# B&R Automation Studio project NAELD004C00R10L518F00 (part 42)

#### Act_Background_QueryWorkOrderInfo.st
```iecst
(** 2021-08-01 **)
ACTION Act_Background_QueryWorkOrderInfo:

	IF eStatus2 <> Error THEN
		IF  uiMilliSecOld <> p_tyDTStructure.millisec THEN
			IF EDGEPOS(p_bLinkOpsMagConvLD1QueryWO) THEN //query false when rcp loaded
				sMagazineId 		:= '1'; //Magazine position to mes
				bGUIDInserted[1]	:= FALSE;
				a_bQueryQueue[i2] 	:= TRUE;
				i2 := i2 + 1;
			ELSIF EDGEPOS(p_bLinkOpsMagConvLD2QueryWO) THEN
				sMagazineId 		:= '2';
				bGUIDInserted[2]	:= FALSE;
				a_bQueryQueue[i2] 	:= TRUE;
				i2 := i2 + 1;
			ELSIF EDGEPOS(p_bLinkOpsMagConvLD3QueryWO) THEN
				sMagazineId 		:= '3';
				bGUIDInserted[3]	:= FALSE;
				a_bQueryQueue[i2] 	:= TRUE;
				i2 := i2 + 1;
			END_IF
		END_IF

//		IF EDGEPOS(p_bQueryWorkOrderInfo) AND p_bAcceptCondition THEN
//		IF (EDGEPOS((p_eLinkCustomerReq = Siemens AND p_bOpsConvWaitForTopUpBrd OR (p_usiLinkProdRcpCurrRcpMcMod = 0 AND bQueryloaderWorkOrder = FALSE) AND bConnected AND p_bOpsRun) AND p_bQueryWorkOrderInfo = FALSE AND bManualQueryWO = FALSE AND p_eLinkCustomerReq = NA)  (*AND p_bAcceptCondition*) AND bReplyWorkOrderInfo= FALSE AND sWorkOrderId = ''))
//			 OR EDGEPOS (p_bQueryWorkOrderInfo) THEN        //Query For Loader           //ADD
//		IF (EDGEPOS((p_bSiemensMcModeChgPrep AND (p_bOpsConvWaitForTopUpBrd OR p_usiLinkProdRcpCurrRcpMcMod = 0)  AND bQueryloaderWorkOrder = FALSE AND bConnected AND p_bOpsRun) AND p_bQueryWorkOrderInfo = FALSE AND bManualQueryWO = FALSE AND bReplyWorkOrderInfo= FALSE AND sWorkOrderId = ''))
//			 OR EDGEPOS (p_bQueryWorkOrderInfo) THEN        //Query For Loader           //ADD
//		IF bQueryloaderWorkOrder = FALSE AND bConnected AND p_bOpsRun AND p_bQueryWorkOrderInfo = FALSE AND bManualQueryWO = FALSE AND bReplyWorkOrderInfo= FALSE AND sWorkOrderId = ''
//			OR EDGEPOS (p_bQueryWorkOrderInfo) THEN        //Query For Loader           //ADD
		IF bQueryloaderWorkOrder = FALSE AND bConnected AND p_bOpsRun AND p_bQueryWorkOrderInfo = FALSE AND bManualQueryWO = FALSE AND bReplyWorkOrderInfo= FALSE AND sWorkOrderId = ''
			OR a_bQueryQueue[0]  THEN
			//OR EDGEPOS (p_bLinkOpsMagConvLD1QueryWO) OR EDGEPOS (p_bLinkOpsMagConvLD2QueryWO) OR EDGEPOS (p_bLinkOpsMagConvLD3QueryWO) THEN        //Query For Loader           //ADD

			fHermesAddOneMsgSend(ADR(a_eMsgSend) , ADR(udiMsgSendBffr) , HermesMsgTypeQueryWorkOrderInfo);

			fHermesGenerateUUID(ADR(tyQueryWorkOrderInfo.tyData.sQueryId) , p_tyDTStructure , pa_usiMacAddr); //Generate QueryID
			uiMilliSecOld :=  p_tyDTStructure.millisec;

			tyQueryWorkOrderInfo.tyData.sMachineId							:= p_sMcId;
			IF sMagazineId = '1'  AND bGUIDInserted[1] = FALSE THEN //Magazine position to mes
				a_MagGUID[1] 		:= tyQueryWorkOrderInfo.tyData.sQueryId;
				bGUIDInserted[1] 	:= TRUE;
			ELSIF sMagazineId = '2' AND bGUIDInserted[2] = FALSE THEN
				a_MagGUID[2] 		:= tyQueryWorkOrderInfo.tyData.sQueryId;
				bGUIDInserted[2] 	:= TRUE;
			ELSIF sMagazineId = '3' AND bGUIDInserted[3] = FALSE THEN
				a_MagGUID[3] 		:= tyQueryWorkOrderInfo.tyData.sQueryId;
				bGUIDInserted[3] 	:= TRUE;
			END_IF

			memcpy(ADR(a_bQueryQueue[0]) , ADR(a_bQueryQueue[1]) , SIZEOF(a_bQueryQueue[0]) * 3);
			a_bQueryQueue[3]	:= FALSE;
			i2 := i2 - 1;

			tyQueryWorkOrderInfo.tyData.sMagazineId							:= p_sMagazineId;
			tyQueryWorkOrderInfo.tyData.iSlotId								:= p_iSlotId;
			tyQueryWorkOrderInfo.tyData.sBarcode						    := p_sBarcode;
			tyQueryWorkOrderInfo.tyAvl.bQueryId							    := tyQueryWorkOrderInfo.tyData.sQueryId <> '';
			tyQueryWorkOrderInfo.tyAvl.bMachineId							:= tyQueryWorkOrderInfo.tyData.sMachineId <> '';
			tyQueryWorkOrderInfo.tyAvl.bMagazineId							:= tyQueryWorkOrderInfo.tyData.sMagazineId <> '';
			tyQueryWorkOrderInfo.tyAvl.bSlotId								:= tyQueryWorkOrderInfo.tyData.iSlotId <> 0;
			tyQueryWorkOrderInfo.tyAvl.bBarcode								:= tyQueryWorkOrderInfo.tyData.sBarcode <> '';

			bQueryloaderWorkOrder := TRUE;
			bRcvWorkOrderInfo1 := FALSE;                     //ADD
			bRcvWorkOrderInfo2 := FALSE;
			bSndWorkOrderInfo  := FALSE;

		END_IF
		                                                                      //Reply Bypass Workorder
//		IF EDGEPOS((p_bSiemensMcModeChgPrep AND bConnected AND p_bOpsRun) AND bReplyBypassWorkOrderInfo= FALSE AND p_bUSHermesUSRdy AND bNewIncomingBoard)  THEN        //Query For Bypass mode           //ADD
//
//
//			fHermesAddOneMsgSend(ADR(a_eMsgSend) , ADR(udiMsgSendBffr) , HermesMsgTypeQueryBypassWOInfo);
//
//			fHermesGenerateUUID(ADR(tyQueryBypassWorkOrderInfo.tyData.sQueryId) , p_tyDTStructure , pa_usiMacAddr); //Generate QueryID
//
//			tyQueryBypassWorkOrderInfo.tyData.sMachineId							:= p_sMcId;
//			tyQueryBypassWorkOrderInfo.tyData.sMagazineId							:= p_sMagazineId;
//			tyQueryBypassWorkOrderInfo.tyData.iSlotId								:= p_iSlotId;
//			tyQueryBypassWorkOrderInfo.tyData.sBarcode						        := sUSBarcode;
//
//			tyQueryBypassWorkOrderInfo.tyAvl.bQueryId							    := tyQueryBypassWorkOrderInfo.tyData.sQueryId <> '';
//			tyQueryBypassWorkOrderInfo.tyAvl.bMachineId						     	:= tyQueryBypassWorkOrderInfo.tyData.sMachineId <> '';
//			tyQueryBypassWorkOrderInfo.tyAvl.bMagazineId							:= tyQueryBypassWorkOrderInfo.tyData.sMagazineId <> '';
//			tyQueryBypassWorkOrderInfo.tyAvl.bSlotId								:= tyQueryBypassWorkOrderInfo.tyData.iSlotId <> 0;
//			tyQueryBypassWorkOrderInfo.tyAvl.bBarcode								:= tyQueryBypassWorkOrderInfo.tyData.sBarcode <> '';
//
//			bQueryBypassWorkOrder := TRUE;
//			bRcvWorkBypassOrderInfo := FALSE;
//			bRcvBypassWorkOrderInfo2 := FALSE;
//			bRcvWorkOrderInfo3      :=FALSE;
//		END_IF

		IF p_bQueryWorkOrderInfo AND p_bAcceptCondition =FALSE THEN
			bRstWorkOrderInfo := TRUE;
		END_IF

		IF tyMsgTypeRcv.bSendWorkOrderInfo THEN

//			IF p_bQueryWorkOrderInfo AND (udiStatus2 = 0) THEN //After CmpParamRcv
//			IF (p_bQueryWorkOrderInfo OR p_bOpsConvWaitForTopUpBrd) AND (udiStatus2 = 0) AND p_tyDI.bTopCoverSWSig THEN //After CmpParamRcv
			IF (p_bQueryWorkOrderInfo OR p_eLinkCustomerReq = Siemens) AND (udiStatus2 = 0) THEN //After CmpParamRcv
				IF tySendWorkOrderInfoRcv.tyAvl.bWorkOrderId AND tySendWorkOrderInfoRcv.tyData.sWorkOrderId <> '' AND
				   tySendWorkOrderInfoRcv.tyData.rWidth >= 50.0 AND tySendWorkOrderInfoRcv.tyData.rWidth <= 460.0	(*AND p_bAcceptCondition*) THEN //Wait Accept Conditon On

					//Priority setting
					memset(ADR(usiSum),0,SIZEOF(usiSum));
					FOR i := 1 TO 3 DO
						usiSum[i]	:= usiSum[i] + usiMagPrior[i];
						IF a_MagGUID[i] = tySendWorkOrderInfoRcv.tyData.sQueryId THEN
							usiSum[i] := usiSum[i] + 10;
						END_IF
					END_FOR
					FOR i1:=1 TO 3 DO
						//Assign Magazine order
						IF  usiSum[i1] >=10 THEN
							IF a_MagAccOrder[1]=0 AND a_MagAccOrder[2]=0 AND a_MagAccOrder[3]=0 THEN
								a_MagAccOrder[i1] := 10; //output
								usiMagOrderPos := i1;
							ELSIF ((a_MagAccOrder[1]=0 AND a_MagAccOrder[2]=0) OR
								(a_MagAccOrder[2]=0 AND a_MagAccOrder[3]=0) OR
								(a_MagAccOrder[1]=0 AND a_MagAccOrder[3]=0)) AND a_MagAccOrder[i1] =0 THEN
								a_MagAccOrder[i1] := 20;
								usiMagOrderPos := i1;
							ELSIF (a_MagAccOrder[1]=0 OR a_MagAccOrder[2]=0 OR a_MagAccOrder[3]=0) AND a_MagAccOrder[i1] =0 THEN
								a_MagAccOrder[i1] := 30;
								usiMagOrderPos := i1;
							END_IF
							bGUIDInserted[i1] := FALSE;
						END_IF
					END_FOR

					bSndWorkOrderInfo  := TRUE;
					bRcvWorkOrderInfo1 := TRUE;
					bRetainNewAcc      := FALSE;                            //ADD
					bQueryloaderWorkOrder := FALSE;
					tySendWorkOrderInfoAcc := tySendWorkOrderInfoRcv;
					tyMsgTypeRcv.bSendWorkOrderInfo := FALSE;
					sWorkOrderId := tySendWorkOrderInfoRcv.tyData.sWorkOrderId;

				ELSIF (tySendWorkOrderInfoRcv.tyAvl.bWorkOrderId = FALSE) OR tySendWorkOrderInfoRcv.tyData.sWorkOrderId = '' OR
					tySendWorkOrderInfoRcv.tyData.rWidth < 50.0 OR tySendWorkOrderInfoRcv.tyData.rWidth > 460.0  THEN
					bRcvWorkOrderInfo2 := TRUE;
					tyMsgTypeRcv.bSendWorkOrderInfo := FALSE;
				END_IF

//			ELSIF p_eLinkCustomerReq = Siemens AND (udiStatus5 = 0) THEN
//				IF tySendWorkOrderInfoRcv.tyAvl.bWorkOrderId AND (tySendWorkOrderInfoRcv.tyData.sWorkOrderId = p_tyUSBoardAvailableRcv.tyData.sWorkOrderId OR tySendWorkOrderInfoRcv.tyData.sWorkOrderId = p_tyUSBoardForecastRcv.tyData.sWorkOrderId) AND
//					tySendWorkOrderInfoRcv.tyAvl.bBatchId AND (tySendWorkOrderInfoRcv.tyData.sBatchId = p_tyUSBoardAvailableRcv.tyData.sBatchId OR tySendWorkOrderInfoRcv.tyData.sBatchId = p_tyUSBoardForecastRcv.tyData.sBatchId) AND
//					tySendWorkOrderInfoRcv.tyAvl.bWidth AND (tySendWorkOrderInfoRcv.tyData.rWidth = p_tyUSBoardAvailableRcv.tyData.rWidth OR tySendWorkOrderInfoRcv.tyData.rWidth = p_tyUSBoardForecastRcv.tyData.rWidth) AND
//					tySendWorkOrderInfoRcv.tyData.rWidth >= 50.0 AND tySendWorkOrderInfoRcv.tyData.rWidth <= 460.0 THEN
//					bRcvWorkBypassOrderInfo := TRUE;
//					tySendBypassWorkOrderInfoAcc := tySendWorkOrderInfoRcv;
//					tyMsgTypeRcv.bSendWorkOrderInfo := FALSE;
//					bRcvWorkOrderInfo3      :=TRUE;
//				ELSE
//					bRcvBypassWorkOrderInfo2 := TRUE;
//					tyMsgTypeRcv.bSendWorkOrderInfo := FALSE;
//				END_IF

			ELSIF p_bQueryWorkOrderInfo = FALSE  THEN
//			ELSIF p_bQueryWorkOrderInfo = FALSE  AND p_bLinkDIPresentSen = FALSE AND ((udiStatus2 = 0) OR (udiStatus5 = 0)) THEN
				tyMsgTypeRcv.bSendWorkOrderInfo := FALSE;
			END_IF
		END_IF

		IF EDGEPOS (bRcvWorkOrderInfo1 = TRUE AND p_bAcceptCondition) THEN

//			tyInfoData1.sProgNm		:= p_sProgNm;
//			tyInfoData1.udiCode		:= 10000;
//			tyInfoData1.eSeverity	:= AlmSeverityInfo;
//			tyInfoData1.sAlmMsg		:= p_sInfoMsg1;

		ELSIF EDGEPOS( bRcvWorkOrderInfo2 = TRUE OR bRcvBypassWorkOrderInfo2) THEN

			tyInfoData2.sProgNm		:= p_sProgNm;
			tyInfoData2.udiCode		:= 10000;
			tyInfoData2.eSeverity	:= AlmSeverityInfo;
			tyInfoData2.sAlmMsg		:= p_sInfoMsg2;

//			bRcvWorkOrderInfo2      := FALSE;
//			bRcvBypassWorkOrderInfo2 := FALSE;

		ELSIF EDGEPOS (bRcvWorkOrderInfo1 = TRUE AND p_bAcceptCondition = FALSE) THEN
//			tyInfoData4.sProgNm		:= p_sProgNm;
//			tyInfoData4.udiCode		:= 10000;
//			tyInfoData4.eSeverity	:= AlmSeverityInfo;
//			tyInfoData4.sAlmMsg		:= p_sInfoMsg4;

		END_IF

//		IF  bRstWorkOrderInfo = TRUE THEN
//
//			tyInfoData3.sProgNm		:= p_sProgNm;
//			tyInfoData3.udiCode		:= 10000;
//			tyInfoData3.eSeverity	:= AlmSeverityInfo;
//			tyInfoData3.sAlmMsg		:= p_sInfoMsg3;	//'Query Work Order Not Possible'
//
//		END_IF

		IF EDGEPOS (bRcvWorkOrderInfo1 OR bRcvWorkOrderInfo2) THEN                       //ReplyWorkOrderInfo for loader

			fHermesAddOneMsgSend(ADR(a_eMsgSend) , ADR(udiMsgSendBffr) , HermesMsgTypeReplyWorkOrderInfo);

			tyReplyWorkOrderInfo.tyData.sWorkOrderId					    := tySendWorkOrderInfoAcc.tyData.sWorkOrderId;
			tyReplyWorkOrderInfo.tyData.sBatchId					      	:= tySendWorkOrderInfoAcc.tyData.sBatchId;
		    IF p_bAcceptCondition AND bRcvWorkOrderInfo2 = FALSE AND p_usiLinkProdRcpCurrRcpMcMod =1  THEN
				tyReplyWorkOrderInfo.tyData.iStatus							    := 1;          //WorkOrder accepted
				bReplyWorkOrderInfo                                             := TRUE;
			ELSIF bRcvWorkOrderInfo2 THEN
				tyReplyWorkOrderInfo.tyData.iStatus							    := 0;         //WorkOrder Rejected
				bReplyWorkOrderInfo                                             := FALSE;
				bRcvWorkOrderInfo2                                              := FALSE;
			ELSE
				tyReplyWorkOrderInfo.tyData.iStatus							    := 2;          //WorkOrder accepted and queue
				bReplyWorkOrderInfo                                             := TRUE;
			END_IF

			tyReplyWorkOrderInfo.tyAvl.bWorkOrderId					:= tySendWorkOrderInfoAcc.tyData.sWorkOrderId <> '';
			tyReplyWorkOrderInfo.tyAvl.bBatchId                     := tySendWorkOrderInfoAcc.tyData.sBatchId <> '';
			tyReplyWorkOrderInfo.tyAvl.bStatus                      :=  TRUE;
			bRcvWorkOrderInfo1 := FALSE;
			bRcvWorkOrderInfo2 := FALSE;

		END_IF

		IF EDGEPOS (bRcvWorkOrderInfo3 OR bRcvBypassWorkOrderInfo2) THEN                       //ReplyWorkOrderInfo for Bypass
			fHermesAddOneMsgSend(ADR(a_eMsgSend) , ADR(udiMsgSendBffr) , HermesMsgTypeReplyWorkOrderInfo);

			tyReplyWorkOrderInfo.tyData.sWorkOrderId					    := tySendBypassWorkOrderInfoAcc.tyData.sWorkOrderId;
			tyReplyWorkOrderInfo.tyData.sBatchId					      	:= tySendBypassWorkOrderInfoAcc.tyData.sBatchId;

			IF p_bAcceptCondition AND p_usiLinkProdRcpCurrRcpMcMod =0 AND bRcvWorkOrderInfo3  THEN
				tyReplyWorkOrderInfo.tyData.iStatus							    := 1;          //WorkOrder accepted
				bReplyBypassWorkOrderInfo                                       := TRUE;
			ELSIF p_bAcceptCondition AND p_usiLinkProdRcpCurrRcpMcMod =1 AND bRcvWorkOrderInfo3 THEN
				tyReplyWorkOrderInfo.tyData.iStatus							    := 2;          //WorkOrder accepted and queue
				bReplyBypassWorkOrderInfo                                       := TRUE;
				bQueryBypassWorkOrder := FALSE;                                               //Add
			ELSIF bRcvBypassWorkOrderInfo2 THEN
				tyReplyWorkOrderInfo.tyData.iStatus							    := 0;          //WorkOrder Rejected
				bReplyBypassWorkOrderInfo                                       := TRUE;
				bRcvBypassWorkOrderInfo2                                        :=FALSE;
			END_IF
			tyReplyWorkOrderInfo.tyAvl.bWorkOrderId					:= tySendWorkOrderInfoAcc.tyData.sWorkOrderId <> '';
			tyReplyWorkOrderInfo.tyAvl.bBatchId                     := tySendWorkOrderInfoAcc.tyData.sBatchId <> '';
			tyReplyWorkOrderInfo.tyAvl.bStatus                      :=  TRUE;
		END_IF

//		IF p_eLinkCustomerReq = Siemens AND p_usiLinkProdRcpCurrRcpMcMod =1 AND  bReplyWorkOrderInfo (*AND p_bLinkDIPresentSen =FALSE*) AND p_tyDI.bConvLftSen = FALSE AND p_tyDI.bConvRgtSen = FALSE (*AND p_tyDI.bTopCoverSWSig*) AND p_bAcceptCondition (*AND p_bUITopUpBrdRdy = FALSE*) THEN   //Add
		IF p_eLinkCustomerReq = Siemens AND  bReplyWorkOrderInfo AND p_tyDI.bConvLftSen = FALSE AND p_tyDI.bConvRgtSen = FALSE AND p_bAcceptCondition THEN   //Add
			bClearWorkOrder := FALSE;
//			tySendWorkOrderInfoNewAcc := tySendWorkOrderInfoAcc;
			tySendWorkOrderInfoNewAcc := tySendWorkOrderInfoRcv;
			diReqWidthInUM	:= REAL_TO_DINT(tySendWorkOrderInfoAcc.tyData.rWidth * 1000);
			p_tyProdRcpCurrRcp.diWidthInUM	:= diReqWidthInUM;
			diReqLoaderWidthInUM := diReqWidthInUM;                 //ADD
			bReplyWorkOrderInfo := FALSE;                           //ADD
			bRetainNewAcc := TRUE;                                  //ADD
			bSendBoardForecast := TRUE;                             //ADD
//		ELSIF p_eLinkCustomerReq = Siemens AND p_usiLinkProdRcpCurrRcpMcMod =0 AND bReplyBypassWorkOrderInfo AND p_bAcceptCondition AND bNewIncomingBoard = FALSE THEN
//			tySendWorkOrderInfoNewAcc := tySendBypassWorkOrderInfoAcc;
//			diReqWidthInUM	:= REAL_TO_DINT(tySendBypassWorkOrderInfoAcc.tyData.rWidth * 1000);
//			IF p_eLinkMcParamUSCommMod = McSetCommModSMEMA THEN
//				p_tyProdRcpCurrRcp.diWidthInUM := diReqLoaderWidthInUM;
//			ELSE
//				p_tyProdRcpCurrRcp.diWidthInUM	:= diReqWidthInUM;
//			END_IF
//			bQueryBypassWorkOrder := FALSE;
//			bReplyBypassWorkOrderInfo := FALSE;
		END_IF

//		IF (p_usiSelProdRcpStep = 1) THEN                         //Standby Bit
//			bClearWorkOrder := TRUE;
//		END_IF

	END_IF

	//		IF p_bQueryWorkOrderInfo = FALSE (*AND p_bLinkDIPresentSen*) AND p_bOpsConvWaitForTopUpBrd= FALSE THEN
	IF  (EDGEPOS(bRcvWorkOrderInfo1 = FALSE AND bRcvWorkOrderInfo2 = FALSE)) THEN
		//Clear Info Message 1
		tyInfoData1.sProgNm		:= '';
		tyInfoData1.udiCode		:= 0;
		tyInfoData1.eSeverity	:= AlmSeverityNA;
		tyInfoData1.sAlmMsg		:= '';
		bRcvWorkOrderInfo1 := FALSE;

		//Clear Info Message 2
		tyInfoData2.sProgNm		:= '';
		tyInfoData2.udiCode		:= 0;
		tyInfoData2.eSeverity	:= AlmSeverityNA;
		tyInfoData2.sAlmMsg		:= '';
		bRcvWorkOrderInfo2 := FALSE;

		//Clear Info Message 3
		tyInfoData3.sProgNm		:= '';
		tyInfoData3.udiCode		:= 0;
		tyInfoData3.eSeverity	:= AlmSeverityNA;
		tyInfoData3.sAlmMsg		:= '';
		bRstWorkOrderInfo := FALSE;

		//Clear Info Message 4
		tyInfoData4.sProgNm		:= '';
		tyInfoData4.udiCode		:= 0;
		tyInfoData4.eSeverity	:= AlmSeverityNA;
		tyInfoData4.sAlmMsg		:= '';
		bRcvWorkOrderInfo1 := FALSE;

	END_IF

//	IF EDGEPOS ((p_bAcceptCondition AND p_eLinkCustomerReq = Siemens AND (p_tyDI.bLoadPosSen OR (p_bLinkStepStackMode  AND p_tyDI.bBrdClrSen= FALSE)) AND p_bOpsConvWaitForTopUpBrd) AND p_usiLinkProdRcpCurrRcpMcMod =1 AND p_bUITopUpBrdRdy = FALSE AND p_bOpsConvTopUpBrdReq = FALSE AND p_tyDI.bBrdStackPresentSen = FALSE AND p_bOpsRun THEN     //Whenever lifter empty clear send work data
//		tySendWorkOrderInfoNewAcc := tyDummySendWorkOrderInfoRcv;
//		sWorkOrderId := '';
//	END_IF

//	IF p_bSendBFId THEN                    //New changeover send Forecast one pulse only
//		bSendBoardForecast := FALSE;
//	END_IF

END_ACTION
```

#### Act_Background_SendBoardArrivedLane1.st
```iecst
(** 2021-08-01 **)
ACTION Act_Background_SendBoardArrivedLane1: //Send after our machine send out "StopTransport" message to upstream

	IF eStatus2 <> Error THEN
		IF tySServiceDescriptionRcv.tyData.tySupportedFeatures.bFeatureBoardTracking = TRUE AND p_tyParam.bFeatureBoardTracking AND bHandshakeDone THEN
			IF EDGEPOS(p_bUSHermesStopTransport1) THEN //p_bConvHvBrd AND p_bPullerRotHmRS;

				fHermesAddOneMsgSend(ADR(a_eMsgSend) , ADR(udiMsgSendBffr) , HermesMsgTypeBoardArrived1);

				tyBoardArrived1.tyData.sMachineId     	        := p_sMcId;
				tyBoardArrived1.tyData.iUpstreamLaneId    	    := p_tyHermesConfiguration.a_tyDSParam[0].iLaneID;
				tyBoardArrived1.tyData.sUpstreamInterfaceId     := p_tyHermesConfiguration.a_tyDSParam[0].sDownstreamInterfaceId;
				tyBoardArrived1.tyData.sMagazineId           	:= sMagPos;//sMagazineId;
				tyBoardArrived1.tyData.iSlotId     	            := iSlotId;
				tyBoardArrived1.tyData.eBoadTransfer    	    := HermesLoaded;
				tyBoardArrived1.tyData.sBoardId     	        := p_sHermesBrdId; //p_tyUSBoardArrived1.tyData.sBoardId;
				tyBoardArrived1.tyData.sBoardIdCreatedBy     	:= p_sMcId; //p_tyUSBoardArrived1.tyData.sBoardIdCreatedBy;
				tyBoardArrived1.tyData.eFailedBoard				:= p_tyAutoRcpTravLif.eFailedBoard; //p_tyUSBoardArrived1.tyData.eFailedBoard;
				tyBoardArrived1.tyData.sProductTypeId			:= p_tyAutoRcpTravLif.sProductTypeId;//p_tyUSBoardArrived1.tyData.sProductTypeId;
				tyBoardArrived1.tyData.eFlippedBoard		  	:= p_tyAutoRcpTravLif.eFlippedBoard;//p_tyUSBoardArrived1.tyData.eFlippedBoard;
				tyBoardArrived1.tyData.sTopBarcode				:= p_tyAutoRcpTravLif.sTopBarcode;//p_tyUSBoardArrived1.tyData.sTopBarcode;
				tyBoardArrived1.tyData.sBottomBarcode			:= p_tyAutoRcpTravLif.sBottomBarcode;//p_tyUSBoardArrived1.tyData.sBottomBarcode;
				tyBoardArrived1.tyData.rLength					:= p_tyAutoRcpTravLif.rLength;//p_tyUSBoardArrived1.tyData.rLength;
				tyBoardArrived1.tyData.rWidth				    := p_tyAutoRcpTravLif.rWidth;//p_tyUSBoardArrived1.tyData.rWidth;
				tyBoardArrived1.tyData.rThickness				:= p_tyAutoRcpTravLif.rThickness;//p_tyUSBoardArrived1.tyData.rThickness;
				tyBoardArrived1.tyData.rConveyorSpeed		    := p_tyAutoRcpTravLif.rConveyorSpeed;//p_tyUSBoardArrived1.tyData.rConveyorSpeed;
				tyBoardArrived1.tyData.rTopClearanceHeight		:= p_tyAutoRcpTravLif.rTopClearanceHeight;//p_tyUSBoardArrived1.tyData.rTopClearanceHeight;
				tyBoardArrived1.tyData.rBottomClearanceHeight	:= p_tyAutoRcpTravLif.rBottomClearanceHeight;//p_tyUSBoardArrived1.tyData.rBottomClearanceHeight;
				tyBoardArrived1.tyData.rWeight					:= p_tyAutoRcpTravLif.rWeight;//p_tyUSBoardArrived1.tyData.rWeight;
				tyBoardArrived1.tyData.sWorkOrdedId             := p_tyAutoRcpTravLif.sWorkOrderId;//p_tyUSBoardArrived1.tyData.sWorkOrderId;
				tyBoardArrived1.tyData.sBatchId                 := p_tyAutoRcpTravLif.sBatchId;//p_tyUSBoardArrived1.tyData.sBatchId;

			    tyBoardArrived1.tyAvl.bMachineId				:= tyBoardArrived1.tyData.sMachineId <> '';
		     	tyBoardArrived1.tyAvl.bUpstreamLaneId			:= tyBoardArrived1.tyData.iUpstreamLaneId <> 0;
		    	tyBoardArrived1.tyAvl.bUpstreamInterfaceId		:= tyBoardArrived1.tyData.sUpstreamInterfaceId <> '';
		    	tyBoardArrived1.tyAvl.bMagazineId		    	:= tyBoardArrived1.tyData.sMagazineId <> '';
		    	tyBoardArrived1.tyAvl.bSlotId				    := tyBoardArrived1.tyData.iSlotId <> 0;
		    	tyBoardArrived1.tyAvl.bBoardTransfer			:= TRUE;
				tyBoardArrived1.tyAvl.bBoardId					:= tyBoardArrived1.tyData.sBoardId <> '';
				tyBoardArrived1.tyAvl.bBoardIdCreatedBy			:= tyBoardArrived1.tyData.sBoardIdCreatedBy <> '';
				tyBoardArrived1.tyAvl.bFailedBoard				:= TRUE;
				tyBoardArrived1.tyAvl.bProductTypeId		  	:= tyBoardArrived1.tyData.sProductTypeId <> '';
				tyBoardArrived1.tyAvl.bFlippedBoard				:= TRUE;
				tyBoardArrived1.tyAvl.bTopBarcode			    := tyBoardArrived1.tyData.sTopBarcode <> '';
				tyBoardArrived1.tyAvl.bBottomBarcode		   	:= tyBoardArrived1.tyData.sBottomBarcode <> '';
				tyBoardArrived1.tyAvl.bLength				    := tyBoardArrived1.tyData.rLength <> 0;
				tyBoardArrived1.tyAvl.bWidth				  	:= tyBoardArrived1.tyData.rWidth <> 0;
				tyBoardArrived1.tyAvl.bThickness			   	:= tyBoardArrived1.tyData.rThickness <> 0;
				tyBoardArrived1.tyAvl.bConveyorSpeed		   	:= tyBoardArrived1.tyData.rConveyorSpeed <> 0;
				tyBoardArrived1.tyAvl.bTopClearanceHeight	    := tyBoardArrived1.tyData.rTopClearanceHeight <> 0;
				tyBoardArrived1.tyAvl.bBottomClearanceHeight    := tyBoardArrived1.tyData.rBottomClearanceHeight <> 0;
		    	tyBoardArrived1.tyAvl.bWeight				    := tyBoardArrived1.tyData.rWeight <> 0;
				tyBoardArrived1.tyAvl.bWorkOrderId				:= tyBoardArrived1.tyData.sWorkOrdedId <> '';
				tyBoardArrived1.tyAvl.bBatchId			    	:= tyBoardArrived1.tyData.sBatchId <> '';

			END_IF

		END_IF

	END_IF

END_ACTION
```

#### Act_Background_SendBoardDepartedLane1.st
```iecst
(** 2021-08-01 **)
ACTION Act_Background_SendBoardDepartedLane1: //Send after our machine send out "TransportFinished" message to downstream

	IF eStatus2 <> Error THEN
		IF tySServiceDescriptionRcv.tyData.tySupportedFeatures.bFeatureBoardTracking = TRUE AND p_tyParam.bFeatureBoardTracking AND bHandshakeDone THEN
			IF EDGEPOS(p_bDSHermesTransportFinished1) THEN

				fHermesAddOneMsgSend(ADR(a_eMsgSend) , ADR(udiMsgSendBffr) , HermesMsgTypeBoardDeparted1);

				tyBoardDeparted1.tyData.sMachineId     	        := p_sMcId;
				tyBoardDeparted1.tyData.iDownstreamLaneId    	:= p_tyHermesConfiguration.a_tyDSParam[0].iLaneID;
				tyBoardDeparted1.tyData.sDownstreamInterfaceId  := p_tyHermesConfiguration.a_tyDSParam[0].sDownstreamInterfaceId;
				tyBoardDeparted1.tyData.sMagazineId           	:= sMagPos;//sMagazineId;
				tyBoardDeparted1.tyData.iSlotId     	        := iSlotId;
				tyBoardDeparted1.tyData.eBoadTransfer    	    := p_eBoardTransfer1;
				tyBoardDeparted1.tyData.sBoardId     	        := p_tyDSBoardDeparted1.tyData.sBoardId;
				tyBoardDeparted1.tyData.sBoardIdCreatedBy     	:= p_tyDSBoardDeparted1.tyData.sBoardIdCreatedBy;
				tyBoardDeparted1.tyData.eFailedBoard			:= p_tyDSBoardDeparted1.tyData.eFailedBoard;
				tyBoardDeparted1.tyData.sProductTypeId			:= p_tyDSBoardDeparted1.tyData.sProductTypeId;
				tyBoardDeparted1.tyData.eFlippedBoard			:= p_tyDSBoardDeparted1.tyData.eFlippedBoard;
				tyBoardDeparted1.tyData.sTopBarcode				:= p_tyDSBoardDeparted1.tyData.sTopBarcode;
				tyBoardDeparted1.tyData.sBottomBarcode			:= p_tyDSBoardDeparted1.tyData.sBottomBarcode;
				tyBoardDeparted1.tyData.rLength					:= p_tyDSBoardDeparted1.tyData.rLength;
				tyBoardDeparted1.tyData.rWidth				    := p_tyDSBoardDeparted1.tyData.rWidth;
				tyBoardDeparted1.tyData.rThickness				:= p_tyDSBoardDeparted1.tyData.rThickness;
				tyBoardDeparted1.tyData.rConveyorSpeed		    := p_tyDSBoardDeparted1.tyData.rConveyorSpeed;
				tyBoardDeparted1.tyData.rTopClearanceHeight		:= p_tyDSBoardDeparted1.tyData.rTopClearanceHeight;
				tyBoardDeparted1.tyData.rBottomClearanceHeight	:= p_tyDSBoardDeparted1.tyData.rBottomClearanceHeight;
				tyBoardDeparted1.tyData.rWeight					:= p_tyDSBoardDeparted1.tyData.rWeight;
				tyBoardDeparted1.tyData.sWorkOrdedId            := p_tyDSBoardDeparted1.tyData.sWorkOrderId;
				tyBoardDeparted1.tyData.sBatchId                := p_tyDSBoardDeparted1.tyData.sBatchId;

				tyBoardDeparted1.tyAvl.bMachineId				:= tyBoardDeparted1.tyData.sMachineId <> '';
				tyBoardDeparted1.tyAvl.bDownstreamLaneId		:= tyBoardDeparted1.tyData.iDownstreamLaneId <> 0;
				tyBoardDeparted1.tyAvl.bDownstreamInterfaceId	:= tyBoardDeparted1.tyData.sDownstreamInterfaceId <> '';
				tyBoardDeparted1.tyAvl.bMagazineId		    	:= tyBoardDeparted1.tyData.sMagazineId <> '';
				tyBoardDeparted1.tyAvl.bSlotId				    := tyBoardDeparted1.tyData.iSlotId <> 0;
				tyBoardDeparted1.tyAvl.bBoardTransfer		    := TRUE;
				tyBoardDeparted1.tyAvl.bBoardId					:= tyBoardDeparted1.tyData.sBoardId <> '';
				tyBoardDeparted1.tyAvl.bBoardIdCreatedBy		:= tyBoardDeparted1.tyData.sBoardIdCreatedBy <> '';
				tyBoardDeparted1.tyAvl.bFailedBoard				:= TRUE;
				tyBoardDeparted1.tyAvl.bProductTypeId		   	:= tyBoardDeparted1.tyData.sProductTypeId <> '';
				tyBoardDeparted1.tyAvl.bFlippedBoard			:= TRUE;
				tyBoardDeparted1.tyAvl.bTopBarcode			    := tyBoardDeparted1.tyData.sTopBarcode <> '';
				tyBoardDeparted1.tyAvl.bBottomBarcode		    := tyBoardDeparted1.tyData.sBottomBarcode <> '';
				tyBoardDeparted1.tyAvl.bLength				    := tyBoardDeparted1.tyData.rLength <> 0;
				tyBoardDeparted1.tyAvl.bWidth				    := (tyBoardDeparted1.tyData.rWidth <> 0);
				tyBoardDeparted1.tyAvl.bThickness			    := (tyBoardDeparted1.tyData.rThickness <> 0);
				tyBoardDeparted1.tyAvl.bConveyorSpeed		    := tyBoardDeparted1.tyData.rConveyorSpeed <> 0;
				tyBoardDeparted1.tyAvl.bTopClearanceHeight	    := (tyBoardDeparted1.tyData.rTopClearanceHeight <> 0);
				tyBoardDeparted1.tyAvl.bBottomClearanceHeight	:= (tyBoardDeparted1.tyData.rBottomClearanceHeight <> 0);
				tyBoardDeparted1.tyAvl.bWeight				    := tyBoardDeparted1.tyData.rWeight <> 0;
				tyBoardDeparted1.tyAvl.bWorkOrderId				:= tyBoardDeparted1.tyData.sWorkOrdedId <> '';
				tyBoardDeparted1.tyAvl.bBatchId			    	:= tyBoardDeparted1.tyData.sBatchId <> '';

			END_IF

		END_IF

	END_IF

END_ACTION
```

#### Act_InitGlobal.st
```iecst
(** 2021-08-01 **)
ACTION Act_InitGlobal:

	(* Always Change If Project Change *)

		//Digital Input
	p_tyDI ACCESS p_DI;

	//Pass Data To Link
	p_bLinkStartupRun ACCESS p_StartupRun;
	p_bLinkOpsMagConvLD1QueryWO ACCESS p_OpsMagConvLD1QueryWO;
	p_bLinkOpsMagConvLD2QueryWO ACCESS p_OpsMagConvLD2QueryWO;
	p_bLinkOpsMagConvLD3QueryWO ACCESS p_OpsMagConvLD3QueryWO;

	//Pass Data To Internal Use
	p_udiRstErr ACCESS p_RstErrReset;
	p_bPrep ACCESS p_NtParamHermesPrep;
	p_tyParam ACCESS p_HermesSvyParam;
	p_sIPAddr ACCESS p_HWInfoIPAddr;
	pa_usiMacAddr ACCESS p_HWInfoMacAddr;
	p_tyDTStructure ACCESS p_TimeCurrDTStruct;
	p_dtCurrDT ACCESS p_TimeCurrDT;
	p_sMcId ACCESS p_McParamMcNm;
	p_sRecipeNm ACCESS p_ProdRcpCurrRcp0Nm;
//	p_sMagazineId ACCESS p_UIMagazineId; // change to mag1,2,3
//	p_iSlotId ACCESS p_UIMagazineSlotId;
	p_sBarcode ACCESS p_UIPCBBarcode;
	p_udiAliveIdleTimeInSec ACCESS p_NtParamSvyHermesAliveTmInSec;
	p_tConnTimeOut ACCESS p_NtParamSvyHermesConnTO;
	p_diTransferInTO ACCESS p_McParamTranOutErrDlyTm;
	p_bNewBrdAvlLastZone ACCESS p_HermesBrdAvlDataNewBrdAvlLastZ;
	p_bOpsRun ACCESS p_OpsRun;
	p_udiFileKeepDay ACCESS p_NtParamSvyHermesFileKeepDay;
	p_sConfigFileName ACCESS p_NtParamSvyHermesConfigFileNm;
	p_sProgNm ACCESS p_NtParamSvyHermesProgNm;
	p_bNtSettingsLoadDone ACCESS p_StartupNtSettingsLoadDone;
	p_bSvyPrep ACCESS p_NtParamHermesSvyPrep;
	p_bSvyEn ACCESS p_McParamHermesSvyEn;
//	p_bQueryWorkOrderInfo ACCESS p_OpsMagConvLD1QueryWO;  //Query WO ****
	p_tyHermesConfiguration ACCESS p_HermesConfiguration;
//	p_bUSHermesStopTransport1 ACCESS p_USHermesStopTransportSnd1; //Lane 1, PCB arrived
//	p_bUSHermesStopTransport2 ACCESS p_USHermesStopTransportSnd2; //Lane 2, open up for specific machine
//	p_bUSHermesStopTransport3 ACCESS p_USHermesStopTransportSnd3; //Lane 3, open up for specific machine
//	p_bUSHermesStopTransport4 ACCESS p_USHermesStopTransportSnd4; //Lane 4, open up for specific machine
//	p_tyUSBoardArrived1 ACCESS p_USHermesBoardArrivedData; //Lane 1
//	p_tyUSBoardArrived2 ACCESS p_USHermesBoardArrivedData2; //Lane 2, open up for specific machine
//	p_tyUSBoardArrived3 ACCESS p_USHermesBoardArrivedData3; //Lane 3, open up for specific machine
//	p_tyUSBoardArrived4 ACCESS p_USHermesBoardArrivedData4; //Lane 4, open up for specific machine
	p_bDSHermesTransportFinished1 ACCESS p_DSHermesATransportFinishedSnd;
//	p_bDSHermesTransportFinished2 ACCESS p_DSHermesTransportFinishedSnd2; //Lane 2, open up for specific machine
//	p_bDSHermesTransportFinished3 ACCESS p_DSHermesTransportFinishedSnd3; //Lane 3, open up for specific machine
//	p_bDSHermesTransportFinished4 ACCESS p_DSHermesTransportFinishedSnd4; //Lane 4, open up for specific machine
	p_tyDSBoardDeparted1 ACCESS p_DSHermesABoardDepartedData; //Lane 1
//	p_tyDSBoardDeparted2 ACCESS p_DSHermesBoardDepartedData2; //Lane 2, open up for specific machine
//	p_tyDSBoardDeparted3 ACCESS p_DSHermesBoardDepartedData3; //Lane 3, open up for specific machine
//	p_tyDSBoardDeparted4 ACCESS p_DSHermesBoardDepartedData4; //Lane 4, open up for specific machine
	p_eHermesStat ACCESS p_HermesStat;
	p_eHermesStatus ACCESS p_HermesStatus;
	p_eMcParamStat ACCESS p_McParamStat;
	p_eMcParamStatus ACCESS p_McParamStatus;
	p_bAllZonesEmpty ACCESS p_DSHermesAAllZonesEmpty; //All zones empty. Before empty, cannot change current sWorkOrderId.
	p_bUIDeleteWorkOrder ACCESS p_UIDeleteWorkOrder;
	p_bAutoRcpCurrDeleteSendWO ACCESS p_AutoRcpCurrDeleteSendWO;
	p_bFirstMcIntheLine ACCESS p_NtParamHermesSvyFirstMc; //First machine in the line only can Query Work Order
	p_sRetainFileName ACCESS p_NtParamSvyHermesRetainFileNm;
	p_tyProdRcpCurrRcp ACCESS p_ProdRcpCurrRcp0;

	p_eLinkCustomerReq ACCESS p_NtParamCustomerReq;          //ADD   Include ReplyWorkOrderID & Machine mode changeover
//	p_bLinkDIPresentSen ACCESS p_DIBrdStackPresentSen;                     //ADD
//	p_bOpsConvTopUpBrdReq ACCESS p_OpsConvTopUpBrdReq;
//	p_bOpsConvWaitForTopUpBrd ACCESS p_OpsConvWaitForTopUpBrd;
//	p_bUITopUpBrdRdy ACCESS p_UITopUpBrdRdy;
	p_bSendBFId ACCESS p_SendBFId;
//	p_usiSelProdRcpStep  ACCESS p_SelProdRcpStep;

	p_usiLinkProdRcpCurrRcpMcMod ACCESS p_ProdRcpCurrRcp0McMod;      //Add
//	p_bUSHermesUSRdy ACCESS p_USHermesUSRdy;
//	pa_tyLinkXMLTableDataBrdAvl1 ACCESS p_USHermesTableDataBrdAvl; //lane 1 B.A
//	p_iLinkXMLTableDataBrdAvlTtlIdx1 ACCESS p_USHermesTableDataBrdAvlTtlIdx; //lane 1 B.A
//	p_tyUSBoardAvailableRcv ACCESS  p_USBoardAvailableRcv;
//	p_tyUSBoardForecastRcv ACCESS p_USBoardForecastRcv;
//	p_bLinkStepStackMode ACCESS p_McParamStepStackMode;

//	p_eLinkMcParamUSCommMod ACCESS p_McParamUSCommMod;
	p_sHermesBrdId ACCESS p_HermesBrdId; //generate for forecast , avail and arrived(supv)

	p_diBuffer1Slt ACCESS p_Buffer1SlotNo;
	p_diBuffer2Slt ACCESS p_Buffer2SlotNo;
	p_diBuffer3Slt ACCESS p_Buffer3SlotNo;

	p_bConvHvBrd ACCESS p_PullConvHvBrd;
	p_bPullerRetRS ACCESS p_DIPullerRetRS;
	p_eOpsTravLifLDPosGo ACCESS p_OpsTravLifLDPosGo;
	p_tyAutoRcpTravLif ACCESS p_AutoRcpTravLif;
	(* Always Change If Project Change *)
END_ACTION
```

#### Act_InitLocal.st
```iecst
(** 2021-08-01 **)
ACTION Act_InitLocal:

	//Input Reference Link To Local Variable
	p_eAct ACCESS ADR(eAct);
	p_udiRstErr ACCESS ADR(udiRstErr);
	p_bPrep ACCESS ADR(bPrep);
	p_bEn ACCESS ADR(bEn);
	p_bDis ACCESS ADR(bDis);
	p_tyParam ACCESS ADR(tyParam);
	p_sIPAddr ACCESS ADR(sIPAddr);
	pa_usiMacAddr ACCESS ADR(a_usiMacAddr);
	p_tyDTStructure ACCESS ADR(tyDTStructure);
	p_dtCurrDT ACCESS ADR(dtCurrDT);
	p_sMcId ACCESS ADR(sMcId);
	p_sMagazineId ACCESS ADR(sMagazineId);
	p_iSlotId ACCESS ADR(iSlotId);
	p_eBoardTransfer1 ACCESS ADR(eBoardTransfer1);
	p_eBoardTransfer2 ACCESS ADR(eBoardTransfer2);
	p_eBoardTransfer3 ACCESS ADR(eBoardTransfer3);
	p_eBoardTransfer4 ACCESS ADR(eBoardTransfer4);
	p_sVersion ACCESS ADR(sVersion);
	p_sBarcode ACCESS ADR(sBarcode);
	p_sRecipeNm ACCESS ADR(sRecipeNm);
	p_udiSndBffrSize ACCESS ADR(udiSndBffrSize);
	p_udiRcvBffrSize ACCESS ADR(udiRcvBffrSize);
	p_udiAliveIdleTimeInSec ACCESS ADR(udiAliveIdleTimeInSec);
	p_tConnTimeOut ACCESS ADR(tConnTimeOut);
	p_diTransferInTO ACCESS ADR(diTransferInTO);
	p_bNewBrdAvlLastZone ACCESS ADR(bNewBrdAvl);
	p_bOpsRun ACCESS ADR(bOpsRun);
	p_udiFileKeepDay ACCESS ADR(udiFileKeepDay);
	p_sConfigFileName ACCESS ADR(sConfigFileName);
	p_sProgNm ACCESS ADR(sProgNm);
	p_bNtSettingsLoadDone ACCESS ADR(bNtSettingsLoadDone);
	p_bSvyPrep ACCESS ADR(bSvyPrep);
	p_bSvyEn ACCESS ADR(bSvyEn);
	p_bQueryWorkOrderInfo ACCESS ADR(bQueryWorkOrderInfo);
	p_tyHermesConfiguration ACCESS ADR(tyHermesCurrConfiguration);
	p_bUSHermesStopTransport1 ACCESS ADR(bUSHermesStopTransportSnd1); //Lane 1
	p_bUSHermesStopTransport2 ACCESS ADR(bUSHermesStopTransportSnd2); //Lane 2
	p_bUSHermesStopTransport3 ACCESS ADR(bUSHermesStopTransportSnd3); //Lane 3
	p_bUSHermesStopTransport4 ACCESS ADR(bUSHermesStopTransportSnd4); //Lane 4
	p_tyUSBoardArrived1 ACCESS ADR(tyUSHermesBoardArrivedData1); //Lane 1
	p_tyUSBoardArrived2 ACCESS ADR(tyUSHermesBoardArrivedData2); //Lane 2
	p_tyUSBoardArrived3 ACCESS ADR(tyUSHermesBoardArrivedData3); //Lane 3
	p_tyUSBoardArrived4 ACCESS ADR(tyUSHermesBoardArrivedData4); //Lane 4
	p_bDSHermesTransportFinished1 ACCESS ADR(bDSHermesTransportFinishedSnd1); //Lane 1
	p_bDSHermesTransportFinished2 ACCESS ADR(bDSHermesTransportFinishedSnd2); //Lane 2
	p_bDSHermesTransportFinished3 ACCESS ADR(bDSHermesTransportFinishedSnd3); //Lane 3
	p_bDSHermesTransportFinished4 ACCESS ADR(bDSHermesTransportFinishedSnd4); //Lane 4
	p_tyDSBoardDeparted1 ACCESS ADR(tyDSHermesBoardDepartedData1); //Lane 1
	p_tyDSBoardDeparted2 ACCESS ADR(tyDSHermesBoardDepartedData2); //Lane 2
	p_tyDSBoardDeparted3 ACCESS ADR(tyDSHermesBoardDepartedData3); //Lane 3
	p_tyDSBoardDeparted4 ACCESS ADR(tyDSHermesBoardDepartedData4); //Lane 4
	p_sInfoMsg ACCESS ADR(sInfoMsg);
	p_sInfoMsg1 ACCESS ADR(sInfoMsg1);
	p_sInfoMsg2 ACCESS ADR(sInfoMsg2);
	p_sInfoMsg3 ACCESS ADR(sInfoMsg3);
	p_sInfoMsg4 ACCESS ADR(sInfoMsg4);
	p_bInternalUse ACCESS ADR(bInternalUse);
	p_sInternalRcv ACCESS ADR(sInternalRcv);
	p_bAcceptCondition ACCESS ADR(bAcceptCondition);
	p_bAllZonesEmpty ACCESS ADR(bAllZonesEmpty);
	p_bDeleteWorkOrder ACCESS ADR(bDeleteWorkOrder);
	p_bFirstMcIntheLine ACCESS ADR(bFirstMcIntheLine);
	p_sRetainFileName ACCESS ADR(sRetainFileName);
	p_udiRetainDataAddr ACCESS ADR(udiRetainDataAddr);
	p_udiRetainDataLen ACCESS ADR(udiRetainDataLen);
	p_sRetainFileName1 ACCESS ADR(sRetainFileName1);           //ADD
	p_sRetainFileName2 ACCESS ADR(sRetainFileName2);
	p_sRetainFileName3 ACCESS ADR(sRetainFileName3);
	p_udiLoaderRetainDataAddr0 ACCESS ADR(udiLoaderRetainDataAddr0);
	p_udiLoaderRetainDataLen0 ACCESS ADR(udiLoaderRetainDataLen0);
	p_udiLoaderRetainDataAddr1 ACCESS ADR(udiLoaderRetainDataAddr1);
	p_udiLoaderRetainDataLen1 ACCESS ADR(udiLoaderRetainDataLen1);
	p_udiBypassRetainDataAddr0 ACCESS ADR(udiBypassRetainDataAddr0);
	p_udiBypassRetainDataLen0 ACCESS ADR(udiBypassRetainDataLen0);        //ADD

END_ACTION
```

#### Act_Link.st
```iecst
(** 2021-08-01 **)
ACTION Act_Link:

	//Board Arrived
	p_bUSHermesStopTransport1 := p_bConvHvBrd AND p_bPullerRetRS;
	IF p_eOpsTravLifLDPosGo = 1 AND p_bConvHvBrd THEN
		sMagPos := '1';
		iSlotId := DINT_TO_INT(p_diBuffer1Slt);
	ELSIF p_eOpsTravLifLDPosGo = 2 AND p_bConvHvBrd THEN
		sMagPos := '2';
		iSlotId := DINT_TO_INT(p_diBuffer2Slt);
	ELSIF p_eOpsTravLifLDPosGo = 3 AND p_bConvHvBrd THEN
		sMagPos := '3';
		iSlotId := DINT_TO_INT(p_diBuffer3Slt);
	END_IF

	//Receive Alive Time
	p_tyParam.tRcvAlive	:= p_tyParam.tSndAlive * 2;

	// For BoardDeparted's BoardTransfer Parameter
	IF p_bFirstMcIntheLine = TRUE AND p_bNewBrdAvlLastZone THEN
		p_eBoardTransfer1 := HermesLoaded;
	ELSIF p_bFirstMcIntheLine = TRUE AND p_bNewBrdAvlLastZone = FALSE THEN
		p_eBoardTransfer1 := HermesLoaded;
	ELSIF p_bFirstMcIntheLine = FALSE AND p_bNewBrdAvlLastZone THEN
		p_eBoardTransfer1 := HermesLoaded;
	ELSIF p_bFirstMcIntheLine = FALSE AND p_bNewBrdAvlLastZone = FALSE THEN
		p_eBoardTransfer1 := HermesLoaded;
	END_IF

	//update magazine mmy
	IF a_MagAccOrder[1]<>0 AND a_MagAccOrder[2]<>0 AND a_MagAccOrder[3]<>0 THEN
	ELSIF a_MagAccOrder[1]<>10 AND a_MagAccOrder[2]<>10 AND a_MagAccOrder[3]<>10 THEN
		FOR i := 1 TO 3 DO
			IF a_MagAccOrder[i] <> 0 THEN
				a_MagAccOrder[i] := a_MagAccOrder[i] -10;
			END_IF
		END_FOR
	END_IF

	//Delete WO
	p_bDeleteWorkOrder := p_bUIDeleteWorkOrder OR p_bAutoRcpCurrDeleteSendWO;

	//Info Message
	p_sInfoMsg		:= 'Hermes Configuration Received From Supervisory System';

	//Info Message 1
	p_sInfoMsg1     := 'Work Order Info Received From Supervisory System';

	//Info Message 2
//	p_sInfoMsg2     := 'Work Order Info Not Found From Supervisory System';
	p_sInfoMsg2     := 'Work Order Or Data Info Invalid From Supervisory System';
	p_sInfoMsg2		:= CONCAT(p_sInfoMsg2 , '$r$n');
	p_sInfoMsg2  	:= CONCAT(p_sInfoMsg2 , 'Please Try Again');

	//Info Message 3
	p_sInfoMsg3     := 'Query Work Order Not Possible';
	p_sInfoMsg3		:= CONCAT(p_sInfoMsg3 , '$r$n');
	p_sInfoMsg3  	:= CONCAT(p_sInfoMsg3 , 'Please Empty the Machines');
	p_sInfoMsg3		:= CONCAT(p_sInfoMsg3 , '$r$n');
	p_sInfoMsg3  	:= CONCAT(p_sInfoMsg3 , 'and Try Again');

	//Info Message 4
	p_sInfoMsg4     := 'Work Order Info Received From Supervisory System';
	p_sInfoMsg4		:= CONCAT(p_sInfoMsg4 , '$r$n');
	p_sInfoMsg4  	:= CONCAT(p_sInfoMsg4 , 'PCB Work Order Info Will Be Queue for next Batch');

	//Accept WorkOrderId from Supervisory System, adjust accordingly
	//(Loader Machine: Magazine area empty, Lifter area empty)
	//(Destacker Machine: load pcb stack area empty and conveyor empty)

	p_bAcceptCondition := p_bAllZonesEmpty; (*AND p_bUITopUpBrdRdy =FALSE*);

//	IF 	p_tyUSBoardAvailableRcv.tyData.sWorkOrderId = '' OR p_tyUSBoardAvailableRcv.tyData.sWorkOrderId <> tySendBypassWorkOrderInfoAcc.tyData.sWorkOrderId OR p_tyUSBoardAvailableRcv.tyData.sBatchId = '' OR  p_tyUSBoardAvailableRcv.tyData.sBatchId <> tySendBypassWorkOrderInfoAcc.tyData.sBatchId OR
//		p_tyUSBoardAvailableRcv.tyData.rWidth = 0 OR p_tyUSBoardAvailableRcv.tyData.rWidth <> tySendBypassWorkOrderInfoAcc.tyData.rWidth THEN
//		IF p_tyUSBoardAvailableRcv.tyData.sTopBarcode <> '' OR p_tyUSBoardAvailableRcv.tyData.sBottomBarcode <> '' THEN
//			sUSBarcode := p_tyUSBoardAvailableRcv.tyData.sTopBarcode;
//			bNewIncomingBoard := TRUE;
//		ELSIF p_tyUSBoardAvailableRcv.tyAvl.bTopBarcode = FALSE OR p_tyUSBoardAvailableRcv.tyAvl.bBottomBarcode THEN
//			sUSBarcode := p_tyUSBoardAvailableRcv.tyData.sBottomBarcode;
//			bNewIncomingBoard := TRUE;
//		ELSE
//			bNewIncomingBoard := FALSE;
//		END_IF
//	ELSIF p_tyUSBoardForecastRcv.tyAvl.bWorkOrderId OR p_tyUSBoardForecastRcv.tyAvl.bBatchId OR p_tyUSBoardForecastRcv.tyAvl.bWeight THEN
//
//		IF p_tyUSBoardForecastRcv.tyData.sWorkOrderId = '' OR p_tyUSBoardForecastRcv.tyData.sWorkOrderId <> tySendBypassWorkOrderInfoAcc.tyData.sWorkOrderId OR p_tyUSBoardForecastRcv.tyData.sBatchId = '' OR  p_tyUSBoardForecastRcv.tyData.sBatchId <> tySendBypassWorkOrderInfoAcc.tyData.sBatchId OR
//			p_tyUSBoardForecastRcv.tyData.rWidth = 0 OR p_tyUSBoardForecastRcv.tyData.rWidth <> tySendBypassWorkOrderInfoAcc.tyData.rWidth THEN
//
//			IF p_tyUSBoardForecastRcv.tyData.sTopBarcode <> '' OR p_tyUSBoardForecastRcv.tyData.sBottomBarcode <> '' THEN
//
//			sUSBarcode := p_tyUSBoardForecastRcv.tyData.sTopBarcode;
//			bNewIncomingBoard := TRUE;
//			ELSIF p_tyUSBoardForecastRcv.tyAvl.bTopBarcode = FALSE OR p_tyUSBoardForecastRcv.tyAvl.bBottomBarcode THEN
//			sUSBarcode := p_tyUSBoardForecastRcv.tyData.sBottomBarcode;
//			bNewIncomingBoard := TRUE;
//			ELSE
//				bNewIncomingBoard := FALSE;
//			END_IF
//		ELSE
//			bNewIncomingBoard := FALSE;
//		END_IF
//	ELSE
//		bNewIncomingBoard := FALSE;
//	END_IF

//	IF EDGENEG (p_bQueryWorkOrderInfo)  THEN
//		IF p_bOpsConvWaitForTopUpBrd THEN
//			bManualQueryWO := TRUE;
//		ELSIF p_bOpsConvWaitForTopUpBrd = FALSE THEN
//			bManualQueryWO := FALSE;
//		END_IF
//	END_IF
//
//	IF p_bOpsConvWaitForTopUpBrd = FALSE THEN
//		bManualQueryWO := FALSE;
//	END_IF

	IF diReqLoaderWidthInUM = 0 THEN                           //Load Data during bootup
		diReqLoaderWidthInUM := REAL_TO_DINT(tySendWorkOrderInfoAcc.tyData.rWidth * 1000);
	END_IF

	IF EDGENEG (p_bLinkStartupRun) THEN
		sWorkOrderId := tySendWorkOrderInfoNewAcc.tyData.sWorkOrderId;
	END_IF

	//	phase 2
//	bChangeOverLifter := lifterEmpty + no UBA + waitTimeOut;
//	bChangeOverLoader := lifterEmpty + UBA + waitTimeOut;
//	IF  p_bAcceptConditionLifter  THEN
//		tySendWorkOrderInfoAccPublish := tySendWorkOrderInfoAcc;
//	ELSIF  p_bAcceptConditionLoader  THEN
//		tySendWorkOrderInfoAccPublish := tySendWorkOrderInfoAcc;
//	END_IF
END_ACTION
```

#### Init.st
```iecst
(** 2021-08-01 **)
PROGRAM _INIT

	(* Always Change If Project Change *)

	//Pass Address To Global Address For External Use
	//Action, State & Status
	p_SvyHermesStat	    	:= ADR(eStat);
	p_SvyHermesStatus   	:= ADR(eMainStatus);
	p_SvyHermesStatTxt    	:= ADR(sStatTxt);
	p_SvyHermesAct	    	:= ADR(eHermesAct);
	p_SvyHermesMcParamAct	:= ADR(eMcParamAct);

	//Alarm
	p_SvyHermesAlmData	    := ADR(tyAlmData);
	p_SvyHermesAlmData1	    := ADR(tyAlmData1);
	p_SvyHermesAlmData2	    := ADR(tyAlmData2);
	p_SvyHermesAlmData3	    := ADR(tyAlmData3);
    p_SvyHermesAlmData4	    := ADR(tyAlmData4);
	p_SvyHermesInfoData	    := ADR(tyInfoData);
	p_SvyHermesInfoData1	:= ADR(tyInfoData1);
	p_SvyHermesInfoData2	:= ADR(tyInfoData2);
	p_SvyHermesInfoData3	:= ADR(tyInfoData3);
	p_SvyHermesInfoData4	:= ADR(tyInfoData4);

	//Output
	p_SvyHermesConnected			:= ADR(bConnected);
	p_SvyHermesHandshakeDone		:= ADR(bHandshakeDone);
	p_SvyHermesInternalSnd		    := ADR(sInternalSnd);
	p_SvyHermesFileNotFound			:= ADR(bFileNotFound);
	p_SvyHermesSetConfiguration	    := ADR(tySetConfigurationModified);
	p_SvyHermesWriteConfig	        := ADR(bWriteConfig);
	p_SvyHermesUpdateUIData	        := ADR(bUpdateUIData);
	p_SvyHermesWorkOrderId          := ADR(sWorkOrderId); //WorkOrderId from Supervisory System
	p_SvyHermesBatchId              := ADR(sBatchId); //BatchId from Supervisory System

	//Data
	p_SvyHermesFoundIndexUS1              := ADR(bFoundIndexUS1);
	p_SvyHermesFoundIndexUS2              := ADR(bFoundIndexUS2);
	p_SvyHermesFoundIndexUS3              := ADR(bFoundIndexUS3);
	p_SvyHermesFoundIndexUS4              := ADR(bFoundIndexUS4);
	p_SvyHermesFoundIndexDS1              := ADR(bFoundIndexDS1);
	p_SvyHermesFoundIndexDS2              := ADR(bFoundIndexDS2);
	p_SvyHermesFoundIndexDS3              := ADR(bFoundIndexDS3);
	p_SvyHermesFoundIndexDS4              := ADR(bFoundIndexDS4);
	p_SvyHermesIndexUS1                   := ADR(udiFoundIndexUS1);
	p_SvyHermesIndexUS2                   := ADR(udiFoundIndexUS2);
	p_SvyHermesIndexUS3                   := ADR(udiFoundIndexUS3);
	p_SvyHermesIndexUS4                   := ADR(udiFoundIndexUS4);
	p_SvyHermesIndexDS1                   := ADR(udiFoundIndexDS1);
	p_SvyHermesIndexDS2                   := ADR(udiFoundIndexDS2);
	p_SvyHermesIndexDS3                   := ADR(udiFoundIndexDS3);
	p_SvyHermesIndexDS4                   := ADR(udiFoundIndexDS4);
	p_RcvBoardInfoOk                      := ADR(bRcvBoardInfoOk);

	//Publish  this to USHermes

	//phase 1
	p_SvyHermesSendWorkOrderDataRcv    := ADR(tySendWorkOrderInfoNewAcc); //from after rcv WO
	p_SvyHermesSendWorkOrderData       := ADR(tySendWorkOrderInfoAcc); //from after send WO
	p_SvyHermesBypassSendWOData        := ADR (tySendBypassWorkOrderInfoAcc);
	p_ReplyWorkOrderInfo               := ADR(bReplyWorkOrderInfo);
	p_SendBoardForecast                := ADR (bSendBoardForecast);
	p_ClearWorkOrder                   := ADR (bClearWorkOrder);
    p_NewIncomingBoard                 := ADR (bNewIncomingBoard);
	p_QueryBypassWorkOrder             := ADR (bQueryBypassWorkOrder);
	p_ReplyBypassWorkOrderInfo         := ADR (bReplyBypassWorkOrderInfo);
	p_ReqLoaderWidthInUM               := ADR  (diReqLoaderWidthInUM);
	p_RcvWorkOrderInfo1                := ADR  (bRcvWorkOrderInfo1);
	p_SndWorkOrderInfo                 := ADR(bSndWorkOrderInfo);

	p_SvyHermesMagAccOrder 			:= ADR(a_MagAccOrder);
	p_SvyHermesMagGUID	 			:= ADR(a_MagGUID);
	p_SvyHermesMagOrderPos 			:= ADR(usiMagOrderPos);
	//phase 2
	//tySendWorkOrderInfoAccPublish
	(* Always Change If Project Change *)

END_PROGRAM
```

### Follower2.var
```iecst
(*2019-06-27*)
(**)
(*Action & State & Status*)
VAR
	p_Follower2Status : UDINT;
END_VAR
(**)
(*Alarm*)
VAR
	p_Follower2AlmData : UDINT;
	p_Follower2InfoData : UDINT;
	p_Follower2InfoData1 : UDINT;
END_VAR
(**)
(*Output*)
VAR
	p_Follower2USAllow : UDINT;
	p_Follower2DSAllow : UDINT;
	p_Follower2ProdAccDataMnl : UDINT;
	p_Follower2ProdUpdtDataMnl : UDINT;
	p_Follower2MagAccDataMnl : UDINT;
	p_Follower2TimeAct : UDINT;
	p_Follower2SetDT : UDINT;
	p_Follower2WaitRlsBrd : UDINT;
	p_Follower2UpdtProdRcp : UDINT;
END_VAR
```

### Program Logical/LF/Follower1

#### InputRef_Link.var
```iecst
(*2019-05-07*)
(**)
VAR
	p_bLinkStartupRun : REFERENCE TO BOOL;
	p_bNtParamAutoRcpPrep : REFERENCE TO BOOL;
	p_eNtParamCustomerReq : REFERENCE TO eCustomer;
END_VAR
(**)
VAR
	p_bLinkOpsRun : REFERENCE TO BOOL;
	p_eLinkNtParamProjMag : REFERENCE TO eLDMag;
	p_bLinkNtParamProjMagConv1Prep : REFERENCE TO BOOL;
	p_bLinkNtParamProjMagConv2Prep : REFERENCE TO BOOL;
	p_bLinkNtParamProjMagConv3Prep : REFERENCE TO BOOL;
	p_bLinkNtParamProjMagConv4Prep : REFERENCE TO BOOL;
	p_bLinkBffr1MagRemoved : REFERENCE TO BOOL;
	p_bLinkBffr2MagRemoved : REFERENCE TO BOOL;
	p_bLinkBffr3MagRemoved : REFERENCE TO BOOL;
	p_bLinkBffr4MagRemoved : REFERENCE TO BOOL;
	p_bLinkOpsMagLD1InitDone : REFERENCE TO BOOL;
	p_bLinkOpsMagLD2InitDone : REFERENCE TO BOOL;
	p_bLinkOpsMagLD3InitDone : REFERENCE TO BOOL;
	p_bLinkOpsMagLD4InitDone : REFERENCE TO BOOL;
	p_bLinkOpsMagConvLD1InitDone : REFERENCE TO BOOL;
	p_bLinkOpsMagConvLD2InitDone : REFERENCE TO BOOL;
	p_bLinkOpsMagConvLD3InitDone : REFERENCE TO BOOL;
	p_bLinkOpsMagConvLD4InitDone : REFERENCE TO BOOL;
END_VAR
(**)
VAR
	bOpsInitDone : BOOL;
	bBffrMagRemoved : BOOL;
END_VAR
(**)
VAR
	p_eLinkUIProdRcpAct : REFERENCE TO eProdRcpAction;
	p_eProdRcpStat : REFERENCE TO eProdRcpAction;
	p_eProdRcpStatus : REFERENCE TO eFBStatus;
	p_tyProdRcpCurrRcpWr : REFERENCE TO tyProdRcpParam;
END_VAR
(**)
VAR
	p_bMcParamMesRFIDEn : REFERENCE TO BOOL;
END_VAR
```

#### Local.var
```iecst
(*2021-05-18*)
(**)
(*Local Action, State & Status*)
VAR
	eStatus : eFBStatus := Idle;
	udiStatus : UDINT := 0;
END_VAR
(**)
(*Local Alarm*)
VAR
	tyAlmData : tyAlmDat;
	tyInfoData : tyAlmDat;
	tyInfoData1 : tyAlmDat;
	a_tyAlmText : ARRAY[10000..10099] OF tyAlmTxt := [(sAlmText:='New Recipe Not Found In Product Recipe List',sRcyText:='Create New Recipe In Product Setting.'),(sAlmText:='Product Recipe Width Not Match',sRcyText:='Check Product Width And Leader Request Width'),(sAlmText:='New Recipe Not Found In Magazine Recipe List',sRcyText:='Create New Recipe In Magazine Setting.'),(sAlmText:='New Recipe Name Empty',sRcyText:='Request Recipe Name From Leader Is Empty, Check Leader Machine'),96(0)];
END_VAR
(**)
(*Local Output*)
VAR
	bUSAllow : BOOL;
	bDSAllow : BOOL;
	bLeaderSeqCtrlInActive : BOOL;
	bProdAccDataMnl : BOOL;
	bProdUpdtDataMnl : BOOL;
	bMagAccDataMnl : BOOL;
	eTimeAct : eTimeAction;
	bWaitRlsBrd : BOOL;
	tyLeaderInfo : tyLFLeaderInfo;
	tyUpdtProdRcp : tyProdRcpParam;
END_VAR
(**)
(*Local Input*)
VAR
	udiRstErr : UDINT := 0;
	bPrep : BOOL := TRUE;
	bEn : BOOL := TRUE;
	bDis : BOOL := FALSE;
	sIPAddr : STRING[15] := '192.168.0.100';
	sMcNm : STRING[30];
	bAWPrep : BOOL := TRUE;
	bAWDis : BOOL;
	bMnlAccData : BOOL;
	bSectionLeader : BOOL;
	sMagRcpNm : STRING[30];
	diWidthLimit : DINT;
	bWidth2Prep : BOOL;
	bUSWidthChkPrep : BOOL;
	bUSWidthChkEn : BOOL;
	bUSWidthChkSen : BOOL;
	bDSWidthChkPrep : BOOL;
	bDSWidthChkEn : BOOL;
	bDSWidthChkSen : BOOL;
	bProdWidthChk : BOOL;
	bUIProdAccData : BOOL;
	bUIProdUpdtData : BOOL;
	bUIMagAccData : BOOL;
	a_tyProdRcpList : ARRAY[1..c_udiProdRcpMax] OF tyProdRcpParam;
	tyCurrProdRcp : tyProdRcpParam;
	sCurrMagRcpNm : STRING[30];
	eTimeStat : eTimeAction;
	eTimeStatus : eFBStatus;
	bAccNewRcpCond : BOOL;
	bUpdtNewRcpCond : BOOL;
	bAutoUpdtData : BOOL;
	sInfoMsg : STRING[200];
	bInternalUse : BOOL;
	tyInternalReqProdRcp : tyProdRcpParam;
	bNewBrdEnteredCond : BOOL;
	bOldBrdExitedCond : BOOL;
	bRlsBrd : BOOL;
	tyToLeaderProdRcp : tyProdRcpParam;
	bInternalReqProdRcpDiff : BOOL;
	bUpdtProdRcpDiff : BOOL;
	bRlsBrdProdRcpDiff : BOOL;
	sProgNm : STRING[15] := 'Follower';
	bNtSettingsLoadDone : BOOL := TRUE;
	tOnlineChkDlyTm : TIME;
	bManual : BOOL := FALSE;
	bErr : BOOL := FALSE;
	bWarning : BOOL := FALSE;
	bOps : BOOL := FALSE;
	bStandby : BOOL := FALSE;
	eAWStat : eAWAction;
END_VAR
(**)
(*Local*)
VAR
	bRstErr : BOOL;
	udiRstErrOld : UDINT;
	bMagAccDataReq1 : BOOL;
	bInitDone : BOOL;
	bInitialDone : BOOL;
	bAutoAccData : BOOL;
	bProdRcpErr : BOOL;
	bMagRcpErr : BOOL;
	bSetTmErr : BOOL;
	bProdAccDataReq : BOOL;
	sReqProdRcpNm : STRING[254];
	diReqProdRcpWidth : DINT;
	bMagAccDataReq : BOOL;
	sReqMagRcpNm : STRING[30];
	usiProdAccDatStep : USINT;
	usiMagAccDatStep : USINT;
	usiProdUpdtDatStep : USINT;
	tyRlsBrdProdRcpNm : tyProdRcpParam;
	bNewBrdEntered : BOOL;
	bOldBrdExited : BOOL;
	i : INT;
	bSetTm : BOOL;
	fbOnlineChk : fbLFFollowerOnlineChk;
	fbFollower : fbLFFollower;
	tyLeaderToFollowerTag : tyLFLeaderToFollowerTag;
	tyFollowerToLeaderTag : tyLFFollowerToLeaderTag;
	eCurrMachineStat : eMachineStat;
	bLeaderOnline : BOOL;
	bLeaderInfo : BOOL;
	bFollowerInfo : BOOL;
	bProdRcpErrNotExist : BOOL;
	bProdRcpErrWidthMismatch : BOOL;
	bDBAOnWOAlign : BOOL;
	udiModuleNum : UDINT := 3901;
END_VAR
```

#### Act_Background_AccData.st
```iecst
(** 2023-02-22 **)
ACTION Act_Background_AccData:
	//Product Accept Data Request
	CASE usiProdAccDatStep OF
		0:
			//Check Error & Request Accept Data
			// If Product Name/Width Error, Check In Background To Update Data
			IF ((eStatus <> Error) AND (bProdAccDataReq = TRUE)) OR bProdRcpErr THEN
				sReqProdRcpNm		:= tyLeaderToFollowerTag.sReqProdRcpNm;
				diReqProdRcpWidth	:= tyLeaderToFollowerTag.diReqProdRcpWidth;
				usiProdAccDatStep	:= 1;
			END_IF

			IF bLeaderOnline=FALSE THEN
				tyInfoData.sProgNm		:= '';
				tyInfoData.udiCode		:= 0;
				tyInfoData.eSeverity	:= AlmSeverityNA;
				tyInfoData.sAlmMsg		:= '';

				bProdRcpErr 			:= FALSE;
				bProdRcpErrNotExist		:= FALSE;
				bProdRcpErrWidthMismatch:= FALSE;
			END_IF

		1:
			IF p_bInternalUse THEN
				usiProdAccDatStep	:= 2;
			ELSE
				//Check In List Of Recipe
				FOR i := 1 TO 2000 DO
					IF sReqProdRcpNm = '' THEN
						EXIT;
					ELSIF sReqProdRcpNm = pa_tyProdRcpList[i].sRcpNm  THEN
						EXIT;
					END_IF
				END_FOR

				IF sReqProdRcpNm = pa_tyProdRcpList[i].sRcpNm AND diReqProdRcpWidth <> pa_tyProdRcpList[i].diWidthInUM THEN
					//Width Mismatch
					bProdRcpErr := TRUE;
					bProdRcpErrWidthMismatch:= TRUE;
					bProdRcpErrNotExist		:= FALSE;
					usiProdAccDatStep	:= 0;
				ELSIF i > 2000 THEN
					//Recipe Not Exist
					bProdRcpErr := TRUE;
					bProdRcpErrNotExist	:= TRUE;
					bProdRcpErrWidthMismatch:= FALSE;
					usiProdAccDatStep	:= 0;
				ELSE
					bProdRcpErr := FALSE;
					bProdRcpErrNotExist	:= FALSE;
					bProdRcpErrWidthMismatch:= FALSE;
					usiProdAccDatStep	:= 2;
				END_IF

				//Info Message
				IF bLeaderOnline=FALSE THEN
					tyInfoData.sProgNm		:= '';
					tyInfoData.udiCode		:= 0;
					tyInfoData.eSeverity	:= AlmSeverityNA;
					tyInfoData.sAlmMsg		:= '';

					bProdRcpErr 			:= FALSE;
					bProdRcpErrNotExist		:= FALSE;
					bProdRcpErrWidthMismatch:= FALSE;
				ELSE

					IF p_bInternalUse = FALSE THEN
						IF bLeaderInfo OR bFollowerInfo THEN
							tyInfoData.sProgNm		:= p_sProgNm;
							tyInfoData.udiCode		:= 10000;
							tyInfoData.eSeverity	:= AlmSeverityInfo;
							tyInfoData.sAlmMsg		:= p_sInfoMsg;
						ELSE
							tyInfoData.sProgNm		:= '';
							tyInfoData.udiCode		:= 0;
							tyInfoData.eSeverity	:= AlmSeverityNA;
							tyInfoData.sAlmMsg		:= '';
						END_IF
					ELSE
						IF p_sInfoMsg <> '' THEN
							tyInfoData.sProgNm		:= p_sProgNm;
							tyInfoData.udiCode		:= 10000;
							tyInfoData.eSeverity	:= AlmSeverityInfo;
							tyInfoData.sAlmMsg		:= p_sInfoMsg;
						ELSE
							tyInfoData.sProgNm		:= '';
							tyInfoData.udiCode		:= 0;
							tyInfoData.eSeverity	:= AlmSeverityNA;
							tyInfoData.sAlmMsg		:= '';
						END_IF

					END_IF
				END_IF
			END_IF
		2:
			//Manual Accept Data Check
			IF bProdAccDataReq = TRUE THEN
				IF bAutoAccData = FALSE THEN
					bProdAccDataMnl	:= TRUE;

					//Info Message
					IF bLeaderOnline=FALSE THEN
						tyInfoData.sProgNm		:= '';
						tyInfoData.udiCode		:= 0;
						tyInfoData.eSeverity	:= AlmSeverityNA;
						tyInfoData.sAlmMsg		:= '';
					ELSE
						IF p_sInfoMsg <> '' THEN
							tyInfoData.sProgNm		:= p_sProgNm;
							tyInfoData.udiCode		:= 10000;
							tyInfoData.eSeverity	:= AlmSeverityInfo;
							tyInfoData.sAlmMsg		:= p_sInfoMsg;
						ELSE
							tyInfoData.sProgNm		:= '';
							tyInfoData.udiCode		:= 0;
							tyInfoData.eSeverity	:= AlmSeverityNA;
							tyInfoData.sAlmMsg		:= '';
						END_IF
					END_IF

					IF p_bUIProdAccData = TRUE THEN
						p_bUIProdAccData := FALSE; //2023_07_26_Debug for Manual Accept Data automatically accept after product change many times
						bProdAccDataMnl		:= FALSE;
						usiProdAccDatStep	:= 3;
					END_IF
				ELSE
					bProdAccDataMnl		:= FALSE;
					usiProdAccDatStep	:= 3;
				END_IF
			ELSE
				bProdAccDataMnl		:= FALSE;
				usiProdAccDatStep	:= 6;
			END_IF

		3:
			//Accept New Recipe Condition
			IF bProdAccDataReq = TRUE THEN
				IF p_bAccNewRcpCond = TRUE THEN

					usiProdAccDatStep	:= 4;
				ELSE
					//Info Message
					IF bLeaderOnline=FALSE THEN
						tyInfoData.sProgNm		:= '';
						tyInfoData.udiCode		:= 0;
						tyInfoData.eSeverity	:= AlmSeverityNA;
						tyInfoData.sAlmMsg		:= '';
					ELSE
						IF p_sInfoMsg <> '' THEN
							tyInfoData.sProgNm		:= p_sProgNm;
							tyInfoData.udiCode		:= 10000;
							tyInfoData.eSeverity	:= AlmSeverityInfo;
							tyInfoData.sAlmMsg		:= p_sInfoMsg;
						ELSE
							tyInfoData.sProgNm		:= '';
							tyInfoData.udiCode		:= 0;
							tyInfoData.eSeverity	:= AlmSeverityNA;
							tyInfoData.sAlmMsg		:= '';
						END_IF
					END_IF
				END_IF
			ELSE
				usiProdAccDatStep	:= 6;
			END_IF

		4:
			//Accept New Recipe Name
			IF p_bInternalUse = TRUE THEN

				p_tyCurrProdRcp	:= p_tyInternalReqProdRcp;
				usiProdAccDatStep := 6;
			ELSE

				FOR i := 1 TO 2000 DO
					IF sReqProdRcpNm = '' THEN
						EXIT;
					ELSIF sReqProdRcpNm = pa_tyProdRcpList[i].sRcpNm THEN
						p_tyCurrProdRcp	:= pa_tyProdRcpList[i];

						EXIT;
					END_IF
				END_FOR

				IF i > 2000 THEN
					//Recipe Not Exist
					bProdRcpErr := TRUE;
					bProdRcpErrNotExist	:= TRUE;
				END_IF
				usiProdAccDatStep	:= 5;
			END_IF

		5:
			(* Add *)
			p_tyProdRcpCurrRcpWr 	:= p_tyCurrProdRcp;
			p_eLinkUIProdRcpAct 	:= ProdRcpActWriteCurrRcpParam;

			IF p_eProdRcpStat = ProdRcpActWriteCurrRcpParam AND p_eProdRcpStatus = Done THEN
				p_eLinkUIProdRcpAct := ProdRcpActIdle;
				usiProdAccDatStep := 6;
			END_IF

		6:
			//Clear Info Message
			tyInfoData.sProgNm		:= '';
			tyInfoData.udiCode		:= 0;
			tyInfoData.eSeverity	:= AlmSeverityNA;
			tyInfoData.sAlmMsg		:= '';

			usiProdAccDatStep	:= 0;

	END_CASE

END_ACTION
```

#### Act_InitGlobal.st
```iecst
(** 2019-06-27 **)
ACTION Act_InitGlobal:

	(* Always Change If Project Change *)

	//Pass Data To Link
	p_bLinkStartupRun ACCESS p_StartupRun;
	p_bNtParamAutoRcpPrep ACCESS p_NtParamAutoRcpPrep;
	p_eNtParamCustomerReq ACCESS p_NtParamCustomerReq;
	p_bMcParamMesRFIDEn ACCESS p_McParamMesRFIDEn;

	p_bLinkOpsRun ACCESS p_OpsRun;
	p_eLinkNtParamProjMag ACCESS p_NtParamProjMag;
	p_bLinkNtParamProjMagConv1Prep ACCESS p_NtParamProjMag1ConvPrep;
	p_bLinkNtParamProjMagConv2Prep ACCESS p_NtParamProjMag2ConvPrep;
	p_bLinkNtParamProjMagConv3Prep ACCESS p_NtParamProjMag3ConvPrep;
	p_bLinkNtParamProjMagConv4Prep ACCESS p_NtParamProjMag4ConvPrep;
	p_bLinkBffr1MagRemoved ACCESS p_Buffer1MagRemoved;
	p_bLinkBffr2MagRemoved ACCESS p_Buffer2MagRemoved;
	p_bLinkBffr3MagRemoved ACCESS p_Buffer3MagRemoved;
	p_bLinkBffr4MagRemoved ACCESS p_Buffer4MagRemoved;
//	p_bLinkOpsMagLD1InitDone ACCESS p_OpsMagLD1InitDone;
//	p_bLinkOpsMagLD2InitDone ACCESS p_OpsMagLD2InitDone;
//	p_bLinkOpsMagLD3InitDone ACCESS p_OpsMagLD3InitDone;
//	p_bLinkOpsMagLD4InitDone ACCESS p_OpsMagLD4InitDone;
	p_bLinkOpsMagConvLD1InitDone ACCESS p_OpsMagConvLD1InitDone;
	p_bLinkOpsMagConvLD2InitDone ACCESS p_OpsMagConvLD2InitDone;
	p_bLinkOpsMagConvLD3InitDone ACCESS p_OpsMagConvLD3InitDone;
	p_bLinkOpsMagConvLD4InitDone ACCESS p_OpsMagConvLD4InitDone;

	//Pass Data To Internal Use
	p_udiRstErr ACCESS p_RstErrReset;
	p_tyCurrProdRcp ACCESS p_ProdRcpCurrRcp1;
//	p_tyInternalReqProdRcp ACCESS p_ProdRcpCurrRcp0;	//Follower 1 Assign With Default Recipe
	p_sProgNm ACCESS p_NtParamFollower1ProgNm;
	p_bNtSettingsLoadDone ACCESS p_StartupNtSettingsLoadDone;

	p_bWidth2Prep ACCESS p_NtParamLFWidth2Prep;

	p_eProdRcpStat ACCESS p_ProdRcpStat; //add
	p_eProdRcpStatus ACCESS p_ProdRcpStatus; //add
	p_eLinkUIProdRcpAct ACCESS p_UIProdRcpAct; //add
	p_tyProdRcpCurrRcpWr ACCESS p_UIProdRcpCurrRcpWr; //add
	(* Always Change If Project Change *)

END_ACTION
```

#### Act_Link.st
```iecst
(** 2019-07-04 **)
ACTION Act_Link:
	IF  p_eNtParamCustomerReq = We_Fabricate AND p_bNtParamAutoRcpPrep  AND p_bMcParamMesRFIDEn THEN
		p_tyInternalReqProdRcp ACCESS p_AutoRcpFollower1;
		p_tyCurrProdRcp	:= p_tyInternalReqProdRcp;
	ELSE
		p_tyInternalReqProdRcp ACCESS p_ProdRcpCurrRcp0;
	END_IF

	//Temporary (Recipe No Save)
	IF p_tyCurrProdRcp.sRcpNm = '' AND p_tyCurrProdRcp.diWidthInUM = 0 THEN
		p_tyCurrProdRcp	:= p_tyInternalReqProdRcp;
	END_IF

	//Info Message
	IF p_eLinkNtParamProjMag = LDMagDual THEN
		bBffrMagRemoved		:= (p_bLinkBffr1MagRemoved = TRUE) AND (p_bLinkBffr2MagRemoved = TRUE);
//		bOpsInitDone		:= ((p_bLinkNtParamProjMagConv1Prep AND p_bLinkOpsMagConvLD1InitDone) OR (NOT p_bLinkNtParamProjMagConv1Prep AND p_bLinkOpsMagLD1InitDone))
//								AND ((p_bLinkNtParamProjMagConv2Prep AND p_bLinkOpsMagConvLD2InitDone) OR (NOT p_bLinkNtParamProjMagConv2Prep AND p_bLinkOpsMagLD2InitDone));
		bOpsInitDone		:= (p_bLinkOpsMagConvLD1InitDone AND p_bLinkOpsMagConvLD2InitDone);
	ELSIF p_eLinkNtParamProjMag = LDMagTriple THEN
		bBffrMagRemoved		:= (p_bLinkBffr1MagRemoved = TRUE) AND (p_bLinkBffr2MagRemoved = TRUE) AND (p_bLinkBffr3MagRemoved = TRUE);
//		bOpsInitDone		:= ((p_bLinkNtParamProjMagConv1Prep AND p_bLinkOpsMagConvLD1InitDone) OR (NOT p_bLinkNtParamProjMagConv1Prep AND p_bLinkOpsMagLD1InitDone))
//								AND ((p_bLinkNtParamProjMagConv2Prep AND p_bLinkOpsMagConvLD2InitDone) OR (NOT p_bLinkNtParamProjMagConv2Prep AND p_bLinkOpsMagLD2InitDone))
//								AND ((p_bLinkNtParamProjMagConv3Prep AND p_bLinkOpsMagConvLD3InitDone) OR (NOT p_bLinkNtParamProjMagConv3Prep AND p_bLinkOpsMagLD3InitDone));
		bOpsInitDone		:= (p_bLinkOpsMagConvLD1InitDone AND p_bLinkOpsMagConvLD2InitDone AND p_bLinkOpsMagConvLD3InitDone);
	ELSIF p_eLinkNtParamProjMag = LDMagQuadruple THEN
		bBffrMagRemoved		:= (p_bLinkBffr1MagRemoved = TRUE) AND (p_bLinkBffr2MagRemoved = TRUE) AND (p_bLinkBffr3MagRemoved = TRUE) AND (p_bLinkBffr4MagRemoved = TRUE);
//		bOpsInitDone		:= ((p_bLinkNtParamProjMagConv1Prep AND p_bLinkOpsMagConvLD1InitDone) OR (NOT p_bLinkNtParamProjMagConv1Prep AND p_bLinkOpsMagLD1InitDone))
//								AND ((p_bLinkNtParamProjMagConv2Prep AND p_bLinkOpsMagConvLD2InitDone) OR (NOT p_bLinkNtParamProjMagConv2Prep AND p_bLinkOpsMagLD2InitDone))
//								AND ((p_bLinkNtParamProjMagConv3Prep AND p_bLinkOpsMagConvLD3InitDone) OR (NOT p_bLinkNtParamProjMagConv3Prep AND p_bLinkOpsMagLD3InitDone))
//								AND ((p_bLinkNtParamProjMagConv4Prep AND p_bLinkOpsMagConvLD4InitDone) OR (NOT p_bLinkNtParamProjMagConv4Prep AND p_bLinkOpsMagLD4InitDone));
		bOpsInitDone		:= p_bLinkOpsMagConvLD1InitDone AND p_bLinkOpsMagConvLD2InitDone AND p_bLinkOpsMagConvLD3InitDone AND p_bLinkOpsMagConvLD4InitDone;
	END_IF

	IF bBffrMagRemoved = FALSE AND p_bNtParamAutoRcpPrep = FALSE THEN
		p_sInfoMsg		:= 'New Recipe Loaded';
		p_sInfoMsg		:= CONCAT(p_sInfoMsg , '$r$n');
		p_sInfoMsg		:= CONCAT(p_sInfoMsg , '$r$n');
		p_sInfoMsg		:= CONCAT(p_sInfoMsg , 'Please Remove All Magazines.');
	ELSE
		p_sInfoMsg		:= '';
	END_IF

	//Accept New Recipe Condition (Before Loaded New Recipe)
	p_bAccNewRcpCond	:= bBffrMagRemoved = TRUE;

	//Update New Recipe Condition (After Loaded New Recipe)
	p_bUpdtNewRcpCond	:= TRUE;

	//Recipe Different
	p_bInternalReqProdRcpDiff	:= memcmp(ADR(p_tyCurrProdRcp) , ADR(p_tyInternalReqProdRcp) , SIZEOF(p_tyCurrProdRcp)) <> 0;
	p_bUpdtProdRcpDiff			:= memcmp(ADR(p_tyCurrProdRcp) , ADR(tyUpdtProdRcp) , SIZEOF(p_tyCurrProdRcp)) <> 0;

END_ACTION
```

#### Act_LinkEn.st
```iecst
(** 2019-04-26 **)
ACTION Act_LinkEn:

	//Link bPrep, bEn & bDis
	p_bDis	:= (p_bLinkStartupRun = TRUE);
//	p_bPrep := p_eNtParamCustomerReq <> We_Fabricate;
END_ACTION
```

### Program Logical/LF/Follower2

#### InputRef_Link.var
```iecst
(*2019-05-07*)
(**)
VAR
	p_bLinkStartupRun : REFERENCE TO BOOL;
	p_bNtParamAutoRcpPrep : REFERENCE TO BOOL;
	p_eNtParamCustomerReq : REFERENCE TO eCustomer;
END_VAR
(**)
VAR
	p_bLinkOpsRun : REFERENCE TO BOOL;
	p_bLinkPullConvHvBrd : REFERENCE TO BOOL;
	p_bLinkOpsTravLifLDInitDone : REFERENCE TO BOOL;
	p_bLinkProjCurtainSenPrep : REFERENCE TO BOOL;
	p_bLinkBypCurtainWidthChg : REFERENCE TO BOOL;
	p_bLinkBypCurtainSenCtrl : REFERENCE TO BOOL;
END_VAR
(**)
VAR
	p_eLinkUIProdRcpAct : REFERENCE TO eProdRcpAction;
	p_eProdRcpStat : REFERENCE TO eProdRcpAction;
	p_eProdRcpStatus : REFERENCE TO eFBStatus;
	p_tyProdRcpCurrRcpWr : REFERENCE TO tyProdRcpParam;
END_VAR
(**)
```

#### Local.var
```iecst
(*2021-05-18*)
(**)
(*Local Action, State & Status*)
VAR
	eStatus : eFBStatus := Idle;
	udiStatus : UDINT := 0;
END_VAR
(**)
(*Local Alarm*)
VAR
	tyAlmData : tyAlmDat;
	tyInfoData : tyAlmDat;
	tyInfoData1 : tyAlmDat;
	a_tyAlmText : ARRAY[10000..10099] OF tyAlmTxt := [(sAlmText:='New Recipe Not Found In Product Recipe List',sRcyText:='Create New Recipe In Product Setting.'),(sAlmText:='Product Recipe Width Not Match',sRcyText:='Check Product Width And Leader Request Width'),(sAlmText:='New Recipe Not Found In Magazine Recipe List',sRcyText:='Create New Recipe In Magazine Setting.'),(sAlmText:='New Recipe Name Empty',sRcyText:='Request Recipe Name From Leader Is Empty, Check Leader Machine'),96(0)];
END_VAR
(**)
(*Local Output*)
VAR
	bUSAllow : BOOL;
	bDSAllow : BOOL;
	bLeaderSeqCtrlInActive : BOOL;
	bProdAccDataMnl : BOOL;
	bProdUpdtDataMnl : BOOL;
	bMagAccDataMnl : BOOL;
	eTimeAct : eTimeAction;
	bWaitRlsBrd : BOOL;
	tyLeaderInfo : tyLFLeaderInfo;
	tyUpdtProdRcp : tyProdRcpParam;
END_VAR
(**)
(*Local Input*)
VAR
	udiRstErr : UDINT := 0;
	bPrep : BOOL := TRUE;
	bEn : BOOL := TRUE;
	bDis : BOOL := FALSE;
	sIPAddr : STRING[15] := '192.168.0.100';
	sMcNm : STRING[30];
	bAWPrep : BOOL := TRUE;
	bAWDis : BOOL;
	bMnlAccData : BOOL;
	bSectionLeader : BOOL;
	sMagRcpNm : STRING[30];
	diWidthLimit : DINT;
	bWidth2Prep : BOOL;
	bUSWidthChkPrep : BOOL;
	bUSWidthChkEn : BOOL;
	bUSWidthChkSen : BOOL;
	bDSWidthChkPrep : BOOL;
	bDSWidthChkEn : BOOL;
	bDSWidthChkSen : BOOL;
	bProdWidthChk : BOOL;
	bUIProdAccData : BOOL;
	bUIProdUpdtData : BOOL;
	bUIMagAccData : BOOL;
	a_tyProdRcpList : ARRAY[1..c_udiProdRcpMax] OF tyProdRcpParam;
	tyCurrProdRcp : tyProdRcpParam;
	sCurrMagRcpNm : STRING[30];
	eTimeStat : eTimeAction;
	eTimeStatus : eFBStatus;
	bAccNewRcpCond : BOOL;
	bUpdtNewRcpCond : BOOL;
	bAutoUpdtData : BOOL;
	sInfoMsg : STRING[200];
	bInternalUse : BOOL;
	tyInternalReqProdRcp : tyProdRcpParam;
	bNewBrdEnteredCond : BOOL;
	bOldBrdExitedCond : BOOL;
	bRlsBrd : BOOL;
	tyToLeaderProdRcp : tyProdRcpParam;
	bInternalReqProdRcpDiff : BOOL;
	bUpdtProdRcpDiff : BOOL;
	bRlsBrdProdRcpDiff : BOOL;
	sProgNm : STRING[15] := 'Follower';
	bNtSettingsLoadDone : BOOL := TRUE;
	tOnlineChkDlyTm : TIME;
	bManual : BOOL := FALSE;
	bErr : BOOL := FALSE;
	bWarning : BOOL := FALSE;
	bOps : BOOL := FALSE;
	bStandby : BOOL := FALSE;
	eAWStat : eAWAction;
END_VAR
(**)
(*Local*)
VAR
	bRstErr : BOOL;
	udiRstErrOld : UDINT;
	bInitDone : BOOL;
	bInitialDone : BOOL;
	bAutoAccData : BOOL;
	bProdRcpErr : BOOL;
	bMagRcpErr : BOOL;
	bSetTmErr : BOOL;
	bProdAccDataReq : BOOL;
	sReqProdRcpNm : STRING[254];
	diReqProdRcpWidth : DINT;
	bMagAccDataReq : BOOL;
	sReqMagRcpNm : STRING[30];
	usiProdAccDatStep : USINT;
	usiMagAccDatStep : USINT;
	usiProdUpdtDatStep : USINT;
	tyRlsBrdProdRcpNm : tyProdRcpParam;
	bNewBrdEntered : BOOL;
	bOldBrdExited : BOOL;
	i : INT;
	bSetTm : BOOL;
	fbOnlineChk : fbLFFollowerOnlineChk;
	fbFollower : fbLFFollower;
	tyLeaderToFollowerTag : tyLFLeaderToFollowerTag;
	tyFollowerToLeaderTag : tyLFFollowerToLeaderTag;
	eCurrMachineStat : eMachineStat;
	bLeaderOnline : BOOL;
	bLeaderInfo : BOOL;
	bSetBffrFull : BOOL;
	bFollowerInfo : BOOL;
	bProdRcpErrNotExist : BOOL;
	bProdRcpErrWidthMismatch : BOOL;
	bDBAOnWOAlign : BOOL;
	udiModuleNum : UDINT := 3901;
END_VAR
```

#### Act_Background.st
```iecst
(** 2021-05-18 **)
ACTION Act_Background:

	IF p_bInternalUse = TRUE THEN
		tyLeaderToFollowerTag.sReqProdRcpNm		:= p_tyInternalReqProdRcp.sRcpNm;
		IF p_bWidth2Prep THEN
			tyLeaderToFollowerTag.diReqProdRcpWidth	:= p_tyInternalReqProdRcp.diWidthInUM2;
		ELSE
			tyLeaderToFollowerTag.diReqProdRcpWidth	:= p_tyInternalReqProdRcp.diWidthInUM;
		END_IF
		tyLeaderToFollowerTag.sReqMagRcpNm		:= '';
		tyLeaderToFollowerTag.bMnlAccData		:= FALSE;
		tyLeaderToFollowerTag.bBypassMnlAccData	:= FALSE;
		tyLeaderToFollowerTag.bBlkDS			:= FALSE;
		tyLeaderToFollowerTag.bBlkUS			:= FALSE;
		tyLeaderToFollowerTag.bBypassWidthChk	:= TRUE;
		tyLeaderToFollowerTag.bSetTm			:= FALSE;
		tyLeaderToFollowerTag.dtTm				:= 0;
		tyLeaderToFollowerTag.uiTmZone			:= 0;
		tyLeaderToFollowerTag.usiRunTm			:= 0;
		tyLeaderToFollowerTag.bProdNameUSWarn	:= FALSE;
		tyLeaderToFollowerTag.bProdNameDSWarn	:= FALSE;
		tyLeaderToFollowerTag.bProdWidthUSWarn	:= FALSE;
		tyLeaderToFollowerTag.bProdWidthDSWarn	:= FALSE;
		tyLeaderToFollowerTag.bLeaderSeqCtrlInActive	:= FALSE;
	END_IF

	Act_Background_UpdtData;

	//FB
	fbFollower.tyLeaderToFollowerTag	:= tyLeaderToFollowerTag;
	fbFollower.sMcNm					:= p_sMcNm;
	fbFollower.sIPAddr					:= p_sIPAddr;
	fbFollower.bSectionLeader			:= p_bSectionLeader;
	fbFollower.sCurrProdRcpNm			:= p_tyCurrProdRcp.sRcpNm;
	fbFollower.diCurrProdWidthUS		:= p_tyCurrProdRcp.diWidthInUM;
	fbFollower.diCurrProdWidthDS		:= p_tyCurrProdRcp.diWidthInUM2;
	fbFollower.sCurrMagRcpNm			:= p_sCurrMagRcpNm;
	fbFollower.sUpdtLeaderProdRcpNm		:= p_tyToLeaderProdRcp.sRcpNm;
	fbFollower.diUpdtLeaderProdWidthUS	:= p_tyToLeaderProdRcp.diWidthInUM;
	fbFollower.diUpdtLeaderProdWidthDS	:= p_tyToLeaderProdRcp.diWidthInUM2;
	fbFollower.sUpdtLeaderMagRcpNm		:= p_sMagRcpNm;
	fbFollower.bMnlAccDat				:= p_bMnlAccData;
	fbFollower.bAWEn					:= (p_bAWPrep = TRUE) AND (p_bAWDis = FALSE);
	fbFollower.bUSWidthChkEn			:= p_bUSWidthChkPrep AND p_bUSWidthChkEn;
	fbFollower.bUSWidthChkSen			:= p_bUSWidthChkSen;
	fbFollower.bDSWidthChkEn			:= p_bDSWidthChkPrep AND p_bDSWidthChkEn;
	fbFollower.bDSWidthChkSen			:= p_bDSWidthChkSen;
	fbFollower.bProdWidthChk			:= p_bProdWidthChk;
	fbFollower.bProdRcpErr				:= bProdRcpErr;
	fbFollower.bMagRcpErr				:= bMagRcpErr;
	fbFollower.bSetTmErr				:= bSetTmErr;
	fbFollower.eCurrMachineStat			:= eCurrMachineStat;
	fbFollower.bProdChgOverActive		:= (p_eAWStat = AWActGoWidthOff);
	fbFollower.bDBAOnWOAlign			:= p_bDBAOnWOAlign;

	fbFollower(bEn := TRUE);

	tyFollowerToLeaderTag	:= fbFollower.tyFollowerToLeaderTag;
	bProdAccDataReq			:= fbFollower.bProdAccDataReq OR (p_bInternalReqProdRcpDiff = TRUE) ;
	bMagAccDataReq			:= fbFollower.bMagAccDataReq;
	bAutoAccData			:= fbFollower.bAutoAccData;

	IF p_bInternalUse THEN
		bLeaderOnline		:= TRUE;
	ELSE
		bLeaderOnline		:= tyLeaderInfo.bOnline;
	END_IF

	IF bLeaderOnline=FALSE THEN
		bUSAllow				:= TRUE;
		bDSAllow				:= TRUE;
		bLeaderSeqCtrlInActive	:= FALSE;
	ELSE
		bUSAllow				:= fbFollower.bUSAllow AND (p_bInternalReqProdRcpDiff = FALSE);;
		bDSAllow				:= fbFollower.bDSAllow;
		bLeaderSeqCtrlInActive	:= tyLeaderToFollowerTag.bLeaderSeqCtrlInActive;
	END_IF

	fbOnlineChk.tyLeaderToFollowerTag	:= tyLeaderToFollowerTag;
	fbOnlineChk(bEn := TRUE);

	Act_Background_AccData;
	Act_Background_ChkRlsBrd;

	//Set Time
	IF EDGEPOS(tyLeaderToFollowerTag.bSetTm) THEN
		bSetTm	:= TRUE;
	END_IF

	IF bSetTm = TRUE THEN
		eTimeAct	:= TimeActSetTime;

		IF (p_eTimeStat = TimeActSetTime) AND (p_eTimeStatus = Done) THEN
			eTimeAct		:= TimeActIdle;
			bSetTm			:= FALSE;
		ELSIF p_eTimeStatus = Error THEN
			eTimeAct		:= TimeActIdle;
			bSetTm			:= FALSE;
		END_IF
	END_IF

	bSetTmErr	:= p_eTimeStatus = Error;

	IF (eStatus = Error) AND bRstErr THEN
		eStatus		:= Idle;
		udiStatus	:= 0;
		bProdRcpErr	:= FALSE;
		bProdRcpErrNotExist	:= FALSE;
		bProdRcpErrWidthMismatch:= FALSE;
		bMagRcpErr	:= FALSE;
	END_IF

END_ACTION
```

#### Act_InitGlobal.st
```iecst
(** 2020-08-06 **)
ACTION Act_InitGlobal:

	(* Always Change If Project Change *)

	//Pass Data To Link
	p_bLinkStartupRun ACCESS p_StartupRun;
	p_bNtParamAutoRcpPrep ACCESS p_NtParamAutoRcpPrep;
	p_eNtParamCustomerReq ACCESS p_NtParamCustomerReq;

	p_bLinkOpsRun ACCESS p_OpsRun;
	p_bLinkPullConvHvBrd ACCESS p_PullConvHvBrd;
	p_bLinkOpsTravLifLDInitDone ACCESS p_OpsTravLifLDInitDone;
	p_bLinkProjCurtainSenPrep ACCESS p_NtParamProjCurtainSenPrep;
	p_bLinkBypCurtainWidthChg ACCESS p_OpsTravLifLBypCurtainWidthChg;
	p_bLinkBypCurtainSenCtrl ACCESS p_OpsTravLifLDBypCurtainSenCtrl;

	//Pass Data To Internal Use
	p_udiRstErr ACCESS p_RstErrReset;
	p_bDSWidthChkPrep ACCESS p_NtParamDSWidthChkPrep;
	p_bDSWidthChkEn ACCESS p_McParamDSWidthChkEn;
	p_bDSWidthChkSen ACCESS p_DIDSWidthChkSen;
	p_tyCurrProdRcp ACCESS p_ProdRcpCurrRcp2;
	p_tyInternalReqProdRcp ACCESS p_Follower1UpdtProdRcp;	//Follower 2 Assign With Follower 1 Recipe
	p_sProgNm ACCESS p_NtParamFollower2ProgNm;
	p_bNtSettingsLoadDone ACCESS p_StartupNtSettingsLoadDone;
	p_bWidth2Prep ACCESS p_NtParamLFWidth2Prep;

	p_eProdRcpStat ACCESS p_ProdRcpStat; //add
	p_eProdRcpStatus ACCESS p_ProdRcpStatus; //add
	p_eLinkUIProdRcpAct ACCESS p_UIProdRcpAct; //add
	p_tyProdRcpCurrRcpWr ACCESS p_UIProdRcpCurrRcpWr; //add
	(* Always Change If Project Change *)

END_ACTION
```

#### Act_InitLocal.st
```iecst
(** 2020-08-06 **)
ACTION Act_InitLocal:

	//Input Reference Link To Local Variable
	p_udiRstErr ACCESS ADR(udiRstErr);
	p_bPrep ACCESS ADR(bPrep);
	p_bEn ACCESS ADR(bEn);
	p_bDis ACCESS ADR(bDis);
	p_sIPAddr ACCESS ADR(sIPAddr);
	p_sMcNm ACCESS ADR(sMcNm);
	p_bAWPrep ACCESS ADR(bAWPrep);
	p_bAWDis ACCESS ADR(bAWDis);
	p_bMnlAccData ACCESS ADR(bMnlAccData);
	p_bSectionLeader ACCESS ADR(bSectionLeader);
	p_sMagRcpNm ACCESS ADR(sMagRcpNm);
	p_diWidthLimit ACCESS ADR(diWidthLimit);
	p_bUSWidthChkPrep ACCESS ADR(bUSWidthChkPrep);
	p_bUSWidthChkEn ACCESS ADR(bUSWidthChkEn);
	p_bUSWidthChkSen ACCESS ADR(bUSWidthChkSen);
	p_bDSWidthChkPrep ACCESS ADR(bDSWidthChkPrep);
	p_bDSWidthChkEn ACCESS ADR(bDSWidthChkEn);
	p_bDSWidthChkSen ACCESS ADR(bDSWidthChkSen);
	p_bProdWidthChk ACCESS ADR(bProdWidthChk);
	p_bUIProdAccData ACCESS ADR(bUIProdAccData);
	p_bUIProdUpdtData ACCESS ADR(bUIProdUpdtData);
	p_bUIMagAccData ACCESS ADR(bUIMagAccData);
	pa_tyProdRcpList ACCESS ADR(a_tyProdRcpList);
	p_tyCurrProdRcp ACCESS ADR(tyCurrProdRcp);
	p_sCurrMagRcpNm ACCESS ADR(sCurrMagRcpNm);
	p_eTimeStat ACCESS ADR(eTimeStat);
	p_eTimeStatus ACCESS ADR(eTimeStatus);
	p_bAccNewRcpCond ACCESS ADR(bAccNewRcpCond);
	p_bUpdtNewRcpCond ACCESS ADR(bUpdtNewRcpCond);
	p_bAutoUpdtData ACCESS ADR(bAutoUpdtData);
	p_sInfoMsg ACCESS ADR(sInfoMsg);
	p_bInternalUse ACCESS ADR(bInternalUse);
	p_tyInternalReqProdRcp ACCESS ADR(tyInternalReqProdRcp);
	p_bNewBrdEnteredCond ACCESS ADR(bNewBrdEnteredCond);
	p_bOldBrdExitedCond ACCESS ADR(bOldBrdExitedCond);
	p_bRlsBrd ACCESS ADR(bRlsBrd);
	p_tyToLeaderProdRcp ACCESS ADR(tyToLeaderProdRcp);
	p_bInternalReqProdRcpDiff ACCESS ADR(bInternalReqProdRcpDiff);
	p_bUpdtProdRcpDiff ACCESS ADR(bUpdtProdRcpDiff);
	p_bRlsBrdProdRcpDiff ACCESS ADR(bRlsBrdProdRcpDiff);
	p_sProgNm ACCESS ADR(sProgNm);
	p_bNtSettingsLoadDone ACCESS ADR(bNtSettingsLoadDone);
	p_tOnlineChkDlyTm ACCESS ADR(tOnlineChkDlyTm);
	p_bManual ACCESS ADR(bManual);
	p_bErr ACCESS ADR(bErr);
	p_bWarning ACCESS ADR(bWarning);
	p_bOps ACCESS ADR(bOps);
	p_bStandby ACCESS ADR(bStandby);
	p_eAWStat ACCESS ADR(eAWStat);
	p_bWidth2Prep ACCESS ADR(bWidth2Prep);
	p_bDBAOnWOAlign ACCESS ADR(bDBAOnWOAlign);

END_ACTION
```

#### Act_Link.st
```iecst
(** 2019-07-04 **)
ACTION Act_Link:
	//Temporary (Recipe No Save)
	IF p_tyCurrProdRcp.sRcpNm = '' AND p_tyCurrProdRcp.diWidthInUM = 0 THEN
		p_tyCurrProdRcp	:= p_tyInternalReqProdRcp;
	END_IF

	//Info Message
	p_sInfoMsg	:= '';

	//Accept New Recipe Condition (Before Loaded New Recipe)
	IF p_bLinkProjCurtainSenPrep = FALSE THEN
		p_bAccNewRcpCond	:= (p_bLinkOpsRun = TRUE) AND (p_bLinkOpsTravLifLDInitDone = TRUE) AND (p_bLinkPullConvHvBrd = FALSE);
	ELSE
		IF p_bLinkBypCurtainSenCtrl THEN
			p_bAccNewRcpCond	:= (p_bLinkOpsRun = TRUE) AND (p_bLinkBypCurtainWidthChg = TRUE) AND (p_bLinkPullConvHvBrd = FALSE);
		ELSE
			p_bAccNewRcpCond	:= (p_bLinkOpsRun = TRUE) AND (p_bLinkOpsTravLifLDInitDone = TRUE) AND (p_bLinkPullConvHvBrd = FALSE);
		END_IF
	END_IF

	//Update New Recipe Condition (After Loaded New Recipe)
	p_bUpdtNewRcpCond	:= TRUE;

	//Recipe Different
	p_bInternalReqProdRcpDiff	:= memcmp(ADR(p_tyCurrProdRcp) , ADR(p_tyInternalReqProdRcp) , SIZEOF(p_tyCurrProdRcp)) <> 0;
	p_bUpdtProdRcpDiff			:= memcmp(ADR(p_tyCurrProdRcp) , ADR(tyUpdtProdRcp) , SIZEOF(p_tyCurrProdRcp)) <> 0;

END_ACTION
```

#### Act_LinkEn.st
```iecst
(** 2019-04-26 **)
ACTION Act_LinkEn:

	//Link bPrep, bEn & bDis
	p_bDis	:= (p_bLinkStartupRun = TRUE);

END_ACTION
```

#### Init.st
```iecst
(** 2019-06-27 **)
PROGRAM _INIT

	(* Always Change If Project Change *)

	//Physical Configuration
	bAutoUpdtData	:= TRUE;
	bInternalUse	:= TRUE;

	//Pass Address To Global Address For External Use
	//Action, State & Status
	p_Follower2Status	:= ADR(eStatus);

	//Alarm
	p_Follower2AlmData		:= ADR(tyAlmData);
	p_Follower2InfoData		:= ADR(tyInfoData);
	p_Follower2InfoData1	:= ADR(tyInfoData1);

	//Output
	p_Follower2USAllow			:= ADR(bUSAllow);
	p_Follower2DSAllow			:= ADR(bDSAllow);
	p_Follower2ProdAccDataMnl	:= ADR(bProdAccDataMnl);
	p_Follower2ProdUpdtDataMnl	:= ADR(bProdUpdtDataMnl);
	p_Follower2MagAccDataMnl	:= ADR(bMagAccDataMnl);
	p_Follower2TimeAct			:= ADR(eTimeAct);
	p_Follower2SetDT			:= ADR(tyLeaderToFollowerTag.dtTm);
	p_Follower2WaitRlsBrd		:= ADR(bWaitRlsBrd);
	p_Follower2UpdtProdRcp		:= ADR(tyUpdtProdRcp);

	(* Always Change If Project Change *)

END_PROGRAM
```

### Program Logical/LF/LFFollower

#### InputRef.var
```iecst
(*2021-05-18*)
(**)
(*General*)
VAR
	p_udiRstErr : REFERENCE TO UDINT;
	p_bPrep : REFERENCE TO BOOL;
	p_bEn : REFERENCE TO BOOL;
	p_bDis : REFERENCE TO BOOL;
END_VAR
(**)
(*Configuration*)
VAR
	p_eAWStat : REFERENCE TO eAWAction;
	p_sIPAddr : REFERENCE TO STRING[15];
END_VAR
(**)
(*Input*)
VAR
	p_sMcNm : REFERENCE TO STRING[30];
	p_bAWPrep : REFERENCE TO BOOL;
	p_bAWDis : REFERENCE TO BOOL;
	p_bMnlAccData : REFERENCE TO BOOL;
	p_bSectionLeader : REFERENCE TO BOOL;
	p_sMagRcpNm : REFERENCE TO STRING[30];
	p_diWidthLimit : REFERENCE TO DINT;
	p_bWidth2Prep : REFERENCE TO BOOL;
	p_bUSWidthChkPrep : REFERENCE TO BOOL;
	p_bUSWidthChkEn : REFERENCE TO BOOL;
	p_bUSWidthChkSen : REFERENCE TO BOOL;
	p_bDSWidthChkPrep : REFERENCE TO BOOL;
	p_bDSWidthChkEn : REFERENCE TO BOOL;
	p_bDSWidthChkSen : REFERENCE TO BOOL;
	p_bProdWidthChk : REFERENCE TO BOOL;
	p_bUIProdAccData : REFERENCE TO BOOL;
	p_bUIProdUpdtData : REFERENCE TO BOOL;
	p_bUIMagAccData : REFERENCE TO BOOL;
	pa_tyProdRcpList : REFERENCE TO ARRAY[1..c_udiProdRcpMax] OF tyProdRcpParam;
	p_tyCurrProdRcp : REFERENCE TO tyProdRcpParam;
	p_tyDispProdRcp : REFERENCE TO tyProdRcpParam;
	p_sCurrMagRcpNm : REFERENCE TO STRING[30];
	p_eTimeStat : REFERENCE TO eTimeAction;
	p_eTimeStatus : REFERENCE TO eFBStatus;
	p_bAccNewRcpCond : REFERENCE TO BOOL;
	p_bUpdtNewRcpCond : REFERENCE TO BOOL;
	p_bAutoUpdtData : REFERENCE TO BOOL;
	p_sInfoMsg : REFERENCE TO STRING[200];
	p_bInternalUse : REFERENCE TO BOOL;
	p_tyInternalReqProdRcp : REFERENCE TO tyProdRcpParam;
	p_bNewBrdEnteredCond : REFERENCE TO BOOL;
	p_bOldBrdExitedCond : REFERENCE TO BOOL;
	p_bRlsBrd : REFERENCE TO BOOL;
	p_tyToLeaderProdRcp : REFERENCE TO tyProdRcpParam;
	p_bInternalReqProdRcpDiff : REFERENCE TO BOOL;
	p_bUpdtProdRcpDiff : REFERENCE TO BOOL;
	p_bRlsBrdProdRcpDiff : REFERENCE TO BOOL;
	p_sProgNm : REFERENCE TO STRING[15];
	p_bNtSettingsLoadDone : REFERENCE TO BOOL;
	p_tOnlineChkDlyTm : REFERENCE TO TIME;
	p_bManual : REFERENCE TO BOOL;
	p_bErr : REFERENCE TO BOOL;
	p_bWarning : REFERENCE TO BOOL;
	p_bOps : REFERENCE TO BOOL;
	p_bStandby : REFERENCE TO BOOL;
	p_bDBAOnWOAlign : REFERENCE TO BOOL;
END_VAR
```

#### InputRef_Link.var
```iecst
(*2023-02-22*)
(**)
VAR
	p_bLinkOpsRun : REFERENCE TO BOOL;
	p_bLinkStartupRun : REFERENCE TO BOOL;
	p_bLinkAWWidthPosDiff : REFERENCE TO BOOL;
	p_bLinkConvBffrLastProduct : REFERENCE TO BOOL;
	p_bLinkBufferLastProductUnload : REFERENCE TO BOOL;
	p_tyLinkBufferBffrStat : REFERENCE TO tyBffrStat;
	p_bLinkNtParamProjLaneBPrep : REFERENCE TO BOOL;
	p_eLinkMcParamDSACommMod : REFERENCE TO eMcSetCommMod;
	p_eLinkMcParamDSBCommMod : REFERENCE TO eMcSetCommMod;
END_VAR
(**)
VAR
	pa_tyMagRcpList : REFERENCE TO ARRAY[1..c_udiMagRcpMax] OF tyMagRcpParam;
	p_tyCurrMagRcp : REFERENCE TO tyMagRcpParam;
END_VAR
(**)
VAR
	sWidthInUMTemp : STRING[80];
	p_eLinkNtParamProjMag : REFERENCE TO eLDMag;
	p_bLinkConvHvBrd : REFERENCE TO BOOL;
	p_bLinkBffr1MagRemoved : REFERENCE TO BOOL;
	p_bLinkBffr2MagRemoved : REFERENCE TO BOOL;
	p_bLinkBffr3MagRemoved : REFERENCE TO BOOL;
END_VAR
(**)
VAR
	p_eLinkUIProdRcpAct : REFERENCE TO eProdRcpAction;
	p_eProdRcpStat : REFERENCE TO eProdRcpAction;
	p_eProdRcpStatus : REFERENCE TO eFBStatus;
	p_tyProdRcpCurrRcpWr : REFERENCE TO tyProdRcpParam;
END_VAR
(**)
```

#### Act_Background.st
```iecst
(** 2021-05-18 **)
ACTION Act_Background:

	IF p_bInternalUse = TRUE THEN
		tyLeaderToFollowerTag.sReqProdRcpNm		:= p_tyInternalReqProdRcp.sRcpNm;
		IF p_bWidth2Prep THEN
			tyLeaderToFollowerTag.diReqProdRcpWidth	:= p_tyInternalReqProdRcp.diWidthInUM2;
		ELSE
			tyLeaderToFollowerTag.diReqProdRcpWidth	:= p_tyInternalReqProdRcp.diWidthInUM;
		END_IF
		tyLeaderToFollowerTag.sReqMagRcpNm		:= '';
		tyLeaderToFollowerTag.bMnlAccData		:= FALSE;
		tyLeaderToFollowerTag.bBypassMnlAccData	:= FALSE;
		tyLeaderToFollowerTag.bBlkDS			:= FALSE;
		tyLeaderToFollowerTag.bBlkUS			:= FALSE;
		tyLeaderToFollowerTag.bBypassWidthChk	:= TRUE;
		tyLeaderToFollowerTag.bSetTm			:= FALSE;
		tyLeaderToFollowerTag.dtTm				:= 0;
		tyLeaderToFollowerTag.uiTmZone			:= 0;
		tyLeaderToFollowerTag.usiRunTm			:= 0;
		tyLeaderToFollowerTag.bProdNameUSWarn	:= FALSE;
		tyLeaderToFollowerTag.bProdNameDSWarn	:= FALSE;
		tyLeaderToFollowerTag.bProdWidthUSWarn	:= FALSE;
		tyLeaderToFollowerTag.bProdWidthDSWarn	:= FALSE;
		tyLeaderToFollowerTag.bLeaderSeqCtrlInActive	:= FALSE;
	END_IF

	Act_Background_UpdtData;

	//FB
	fbFollower.tyLeaderToFollowerTag	:= tyLeaderToFollowerTag;
	fbFollower.sMcNm					:= p_sMcNm;
	fbFollower.sIPAddr					:= p_sIPAddr;
	fbFollower.bSectionLeader			:= p_bSectionLeader;
	fbFollower.sCurrProdRcpNm			:= p_tyCurrProdRcp.sRcpNm;
	fbFollower.diCurrProdWidthUS		:= p_tyCurrProdRcp.diWidthInUM;
	fbFollower.diCurrProdWidthDS		:= p_tyCurrProdRcp.diWidthInUM2;
	fbFollower.sCurrMagRcpNm			:= p_sCurrMagRcpNm;
	fbFollower.sUpdtLeaderProdRcpNm		:= p_tyToLeaderProdRcp.sRcpNm;
	fbFollower.diUpdtLeaderProdWidthUS	:= p_tyToLeaderProdRcp.diWidthInUM;
	fbFollower.diUpdtLeaderProdWidthDS	:= p_tyToLeaderProdRcp.diWidthInUM2;
	fbFollower.sUpdtLeaderMagRcpNm		:= p_sMagRcpNm;
	fbFollower.bMnlAccDat				:= p_bMnlAccData;
	fbFollower.bAWEn					:= (p_bAWPrep = TRUE) AND (p_bAWDis = FALSE);
	fbFollower.bUSWidthChkEn			:= p_bUSWidthChkPrep AND p_bUSWidthChkEn;
	fbFollower.bUSWidthChkSen			:= p_bUSWidthChkSen;
	fbFollower.bDSWidthChkEn			:= p_bDSWidthChkPrep AND p_bDSWidthChkEn;
	fbFollower.bDSWidthChkSen			:= p_bDSWidthChkSen;
	fbFollower.bProdWidthChk			:= p_bProdWidthChk;
	fbFollower.bProdRcpErr				:= bProdRcpErr;
	fbFollower.bMagRcpErr				:= bMagRcpErr;
	fbFollower.bSetTmErr				:= bSetTmErr;
	fbFollower.eCurrMachineStat			:= eCurrMachineStat;
	fbFollower.bProdChgOverActive		:= (p_eAWStat = AWActGoWidthOff);
	fbFollower.bDBAOnWOAlign			:= p_bDBAOnWOAlign;

	fbFollower(bEn := TRUE);

	tyFollowerToLeaderTag	:= fbFollower.tyFollowerToLeaderTag;
	bProdAccDataReq			:= fbFollower.bProdAccDataReq OR (p_bInternalReqProdRcpDiff = TRUE) ;
	bMagAccDataReq			:= fbFollower.bMagAccDataReq;
	bAutoAccData			:= fbFollower.bAutoAccData;

	bLeaderOnline			:= tyLeaderInfo.bOnline;

	IF bLeaderOnline=FALSE THEN
		bUSAllow				:= TRUE;
		bDSAllow				:= TRUE;
		bLeaderSeqCtrlInActive	:= FALSE;
	ELSE
		bUSAllow				:= fbFollower.bUSAllow AND (p_bInternalReqProdRcpDiff = FALSE);;
		bDSAllow				:= fbFollower.bDSAllow;
		bLeaderSeqCtrlInActive	:= tyLeaderToFollowerTag.bLeaderSeqCtrlInActive;
	END_IF

	fbOnlineChk.tyLeaderToFollowerTag	:= tyLeaderToFollowerTag;
	fbOnlineChk(bEn := TRUE);

	Act_Background_AccData;
	Act_Background_ChkRlsBrd;

	//Set Time
	IF EDGEPOS(tyLeaderToFollowerTag.bSetTm) THEN
		bSetTm	:= TRUE;
	END_IF

	IF bSetTm = TRUE THEN
		eTimeAct	:= TimeActSetTime;

		IF (p_eTimeStat = TimeActSetTime) AND (p_eTimeStatus = Done) THEN
			eTimeAct		:= TimeActIdle;
			bSetTm			:= FALSE;
		ELSIF p_eTimeStatus = Error THEN
			eTimeAct		:= TimeActIdle;
			bSetTm			:= FALSE;
		END_IF
	END_IF

	bSetTmErr	:= p_eTimeStatus = Error;

	IF (eStatus = Error) AND bRstErr THEN
		eStatus		:= Idle;
		udiStatus	:= 0;
		bProdRcpErr	:= FALSE;
		bProdRcpErrNotExist	:= FALSE;
		bProdRcpErrWidthMismatch:= FALSE;
		bMagRcpErr	:= FALSE;
	END_IF

END_ACTION
```

#### Act_Background_AccData.st
```iecst
(** 2023-02-22 **)
ACTION Act_Background_AccData:
	//Product Accept Data Request
	CASE usiProdAccDatStep OF
		0:
			//Check Error & Request Accept Data
			// If Product Name/Width Error, Check In Background To Update Data
			IF ((eStatus <> Error) AND (bProdAccDataReq = TRUE)) OR bProdRcpErr THEN
				sReqProdRcpNm		:= tyLeaderToFollowerTag.sReqProdRcpNm;
				diReqProdRcpWidth	:= tyLeaderToFollowerTag.diReqProdRcpWidth;
				usiProdAccDatStep	:= 1;
			END_IF

			IF bLeaderOnline=FALSE THEN
				tyInfoData.sProgNm		:= '';
				tyInfoData.udiCode		:= 0;
				tyInfoData.eSeverity	:= AlmSeverityNA;
				tyInfoData.sAlmMsg		:= '';

				bProdRcpErr 			:= FALSE;
				bProdRcpErrNotExist		:= FALSE;
				bProdRcpErrWidthMismatch:= FALSE;
			END_IF

		1:
			IF p_bInternalUse THEN
				usiProdAccDatStep	:= 2;
			ELSE
				//Check In List Of Recipe
				FOR i := 1 TO 2000 DO
					IF sReqProdRcpNm = '' THEN
						EXIT;
					ELSIF sReqProdRcpNm = pa_tyProdRcpList[i].sRcpNm  THEN
						EXIT;
					END_IF
				END_FOR

				IF sReqProdRcpNm = pa_tyProdRcpList[i].sRcpNm AND diReqProdRcpWidth <> pa_tyProdRcpList[i].diWidthInUM THEN
					//Width Mismatch
					bProdRcpErr := TRUE;
					bProdRcpErrWidthMismatch:= TRUE;
					bProdRcpErrNotExist		:= FALSE;
					usiProdAccDatStep	:= 0;
				ELSIF i > 2000 THEN
					//Recipe Not Exist
					bProdRcpErr := TRUE;
					bProdRcpErrNotExist	:= TRUE;
					bProdRcpErrWidthMismatch:= FALSE;
					usiProdAccDatStep	:= 0;
				ELSE
					bProdRcpErr := FALSE;
					bProdRcpErrNotExist	:= FALSE;
					bProdRcpErrWidthMismatch:= FALSE;
					usiProdAccDatStep	:= 2;
				END_IF

				//Info Message
				IF bLeaderOnline=FALSE THEN
					tyInfoData.sProgNm		:= '';
					tyInfoData.udiCode		:= 0;
					tyInfoData.eSeverity	:= AlmSeverityNA;
					tyInfoData.sAlmMsg		:= '';

					bProdRcpErr 			:= FALSE;
					bProdRcpErrNotExist		:= FALSE;
					bProdRcpErrWidthMismatch:= FALSE;
				ELSE

					IF p_bInternalUse = FALSE THEN
						IF bLeaderInfo OR bFollowerInfo THEN
							tyInfoData.sProgNm		:= p_sProgNm;
							tyInfoData.udiCode		:= 10000;
							tyInfoData.eSeverity	:= AlmSeverityInfo;
							tyInfoData.sAlmMsg		:= p_sInfoMsg;
						ELSE
							tyInfoData.sProgNm		:= '';
							tyInfoData.udiCode		:= 0;
							tyInfoData.eSeverity	:= AlmSeverityNA;
							tyInfoData.sAlmMsg		:= '';
						END_IF
					ELSE
						IF p_sInfoMsg <> '' THEN
							tyInfoData.sProgNm		:= p_sProgNm;
							tyInfoData.udiCode		:= 10000;
							tyInfoData.eSeverity	:= AlmSeverityInfo;
							tyInfoData.sAlmMsg		:= p_sInfoMsg;
						ELSE
							tyInfoData.sProgNm		:= '';
							tyInfoData.udiCode		:= 0;
							tyInfoData.eSeverity	:= AlmSeverityNA;
							tyInfoData.sAlmMsg		:= '';
						END_IF

					END_IF
				END_IF
			END_IF
		2:
			//Manual Accept Data Check
			IF bProdAccDataReq = TRUE THEN
				IF bAutoAccData = FALSE THEN
					bProdAccDataMnl	:= TRUE;

					//Info Message
					IF bLeaderOnline=FALSE THEN
						tyInfoData.sProgNm		:= '';
						tyInfoData.udiCode		:= 0;
						tyInfoData.eSeverity	:= AlmSeverityNA;
						tyInfoData.sAlmMsg		:= '';
					ELSE
						IF p_sInfoMsg <> '' THEN
							tyInfoData.sProgNm		:= p_sProgNm;
							tyInfoData.udiCode		:= 10000;
							tyInfoData.eSeverity	:= AlmSeverityInfo;
							tyInfoData.sAlmMsg		:= p_sInfoMsg;
						ELSE
							tyInfoData.sProgNm		:= '';
							tyInfoData.udiCode		:= 0;
							tyInfoData.eSeverity	:= AlmSeverityNA;
							tyInfoData.sAlmMsg		:= '';
						END_IF
					END_IF

					IF p_bUIProdAccData = TRUE THEN
						p_bUIProdAccData := FALSE; //2023_07_26_Debug for Manual Accept Data automatically accept after product change many times
						bProdAccDataMnl		:= FALSE;
						usiProdAccDatStep	:= 3;
					END_IF
				ELSE
					p_bUIProdAccData := FALSE; //2023_07_26_Debug for Manual Accept Data automatically accept after product change many times
					bProdAccDataMnl		:= FALSE;
					usiProdAccDatStep	:= 3;
				END_IF
			ELSE
				bProdAccDataMnl		:= FALSE;
				usiProdAccDatStep	:= 6;
			END_IF

		3:
			//Accept New Recipe Condition
			IF bProdAccDataReq = TRUE THEN
				IF p_bAccNewRcpCond = TRUE THEN

					usiProdAccDatStep	:= 4;
				ELSE
					//Info Message
					IF bLeaderOnline=FALSE THEN
						tyInfoData.sProgNm		:= '';
						tyInfoData.udiCode		:= 0;
						tyInfoData.eSeverity	:= AlmSeverityNA;
						tyInfoData.sAlmMsg		:= '';
					ELSE
						IF p_sInfoMsg <> '' THEN
							tyInfoData.sProgNm		:= p_sProgNm;
							tyInfoData.udiCode		:= 10000;
							tyInfoData.eSeverity	:= AlmSeverityInfo;
							tyInfoData.sAlmMsg		:= p_sInfoMsg;
						ELSE
							tyInfoData.sProgNm		:= '';
							tyInfoData.udiCode		:= 0;
							tyInfoData.eSeverity	:= AlmSeverityNA;
							tyInfoData.sAlmMsg		:= '';
						END_IF
					END_IF
				END_IF
			ELSE
				usiProdAccDatStep	:= 6;
			END_IF

		4:
			//Accept New Recipe Name
			IF p_bInternalUse = TRUE THEN

				p_tyCurrProdRcp	:= p_tyInternalReqProdRcp;
				usiProdAccDatStep := 6;
			ELSE

				FOR i := 1 TO 2000 DO
					IF sReqProdRcpNm = '' THEN
						EXIT;
					ELSIF sReqProdRcpNm = pa_tyProdRcpList[i].sRcpNm THEN
						p_tyCurrProdRcp	:= pa_tyProdRcpList[i];

						EXIT;
					END_IF
				END_FOR

				IF i > 2000 THEN
					//Recipe Not Exist
					bProdRcpErr := TRUE;
					bProdRcpErrNotExist	:= TRUE;
				END_IF
				usiProdAccDatStep	:= 5;
			END_IF

		5:
			(* Add *)
			p_tyProdRcpCurrRcpWr 	:= p_tyCurrProdRcp;
			p_eLinkUIProdRcpAct 	:= ProdRcpActWriteCurrRcpParam;

			IF p_eProdRcpStat = ProdRcpActWriteCurrRcpParam AND p_eProdRcpStatus = Done THEN
				p_eLinkUIProdRcpAct := ProdRcpActIdle;
				usiProdAccDatStep := 6;
			END_IF

		6:
			//Clear Info Message
			tyInfoData.sProgNm		:= '';
			tyInfoData.udiCode		:= 0;
			tyInfoData.eSeverity	:= AlmSeverityNA;
			tyInfoData.sAlmMsg		:= '';

			usiProdAccDatStep	:= 0;

	END_CASE

END_ACTION
```

#### Act_InitGlobal.st
```iecst
(** 2023-02-22 **)
ACTION Act_InitGlobal:

	(* Always Change If Project Change *)

	//Pass Data To Link
	p_bLinkStartupRun ACCESS p_StartupRun;
	p_bLinkOpsRun ACCESS p_OpsRun;

	p_eLinkNtParamProjMag ACCESS p_NtParamProjMag;
	p_bLinkConvHvBrd ACCESS p_PullConvHvBrd;
	p_bLinkBffr1MagRemoved ACCESS p_Buffer1MagRemoved;
	p_bLinkBffr2MagRemoved ACCESS p_Buffer2MagRemoved;
	p_bLinkBffr3MagRemoved ACCESS p_Buffer3MagRemoved;

	//Pass Data To Internal Use
	p_udiRstErr ACCESS p_RstErrReset;
	p_bPrep ACCESS p_NtParamLFPrep;
	p_bEn ACCESS p_McParamLFEn;
	p_sIPAddr ACCESS p_HWInfoIPAddr;
	p_sMcNm ACCESS p_McParamMcNm;
	p_bAWPrep ACCESS p_NtParamAWPrep;
	p_bAWDis ACCESS p_McParamAWDis;
	p_bMnlAccData ACCESS p_McParamMnlAccDat;
	p_bSectionLeader ACCESS p_McParamSectionLeader;
	p_diWidthLimit ACCESS p_NtParamLFWidthLimit;
	p_bProdWidthChk ACCESS p_NtParamLFProdWidthChk;
	p_bUIProdAccData ACCESS p_UIProdAccData;
	p_bUIMagAccData ACCESS p_UIMagAccData;
	pa_tyProdRcpList ACCESS p_ProdRcpCurrList;
	p_tyCurrProdRcp ACCESS p_ProdRcpCurrRcp0;
	p_tyDispProdRcp ACCESS p_ProdRcpCurrRcp1;
//	p_sCurrMagRcpNm ACCESS ADR(p_tyCurrMagRcp.sRcpNm);
	p_eTimeStat ACCESS p_TimeStat;
	p_eTimeStatus ACCESS p_TimeStatus;
	p_tyToLeaderProdRcp ACCESS p_Follower2UpdtProdRcp;	//Assign With Conveyor Last Zone (To Leader Completion Update)
	p_sProgNm ACCESS p_NtParamLFFollowerProgNm;
	p_bNtSettingsLoadDone ACCESS p_StartupNtSettingsLoadDone;

	p_tOnlineChkDlyTm ACCESS p_NtParamLFFllowerOnlineChkDlyTm;
	p_bManual ACCESS p_UIUIMnlMod;
	p_bErr ACCESS p_AlarmErr;
	p_bOps ACCESS p_OpsStatusRun;
	p_bStandby ACCESS p_OpsStatusStop;
	p_bWarning ACCESS p_AlarmWarning;
	p_eAWStat ACCESS p_AWOpenStat;
	p_bWidth2Prep ACCESS p_NtParamLFWidth2Prep;

	p_bLinkNtParamProjLaneBPrep ACCESS p_NtParamProjLaneBPrep;
	p_eLinkMcParamDSACommMod ACCESS p_McParamDSCommAMod;
	p_eLinkMcParamDSBCommMod ACCESS p_McParamDSCommBMod;

	p_bDBAOnWOAlign ACCESS p_McParamDBAOnWOAlign;

	p_eProdRcpStat ACCESS p_ProdRcpStat; //add
	p_eProdRcpStatus ACCESS p_ProdRcpStatus; //add
	p_eLinkUIProdRcpAct ACCESS p_UIProdRcpAct; //add
	p_tyProdRcpCurrRcpWr ACCESS p_UIProdRcpCurrRcpWr; //add

	(* Always Change If Project Change *)

END_ACTION
```

#### Act_InitLocal.st
```iecst
(** 2021-05-18 **)
ACTION Act_InitLocal:

	//Input Reference Link To Local Variable
	p_udiRstErr ACCESS ADR(udiRstErr);
	p_bPrep ACCESS ADR(bPrep);
	p_bEn ACCESS ADR(bEn);
	p_bDis ACCESS ADR(bDis);
	p_sIPAddr ACCESS ADR(sIPAddr);
	p_sMcNm ACCESS ADR(sMcNm);
	p_bAWPrep ACCESS ADR(bAWPrep);
	p_bAWDis ACCESS ADR(bAWDis);
	p_bMnlAccData ACCESS ADR(bMnlAccData);
	p_bSectionLeader ACCESS ADR(bSectionLeader);
	p_sMagRcpNm ACCESS ADR(sMagRcpNm);
	p_diWidthLimit ACCESS ADR(diWidthLimit);
	p_bUSWidthChkPrep ACCESS ADR(bUSWidthChkPrep);
	p_bUSWidthChkEn ACCESS ADR(bUSWidthChkEn);
	p_bUSWidthChkSen ACCESS ADR(bUSWidthChkSen);
	p_bDSWidthChkPrep ACCESS ADR(bDSWidthChkPrep);
	p_bDSWidthChkEn ACCESS ADR(bDSWidthChkEn);
	p_bDSWidthChkSen ACCESS ADR(bDSWidthChkSen);
	p_bProdWidthChk ACCESS ADR(bProdWidthChk);
	p_bUIProdAccData ACCESS ADR(bUIProdAccData);
	p_bUIProdUpdtData ACCESS ADR(bUIProdUpdtData);
	p_bUIMagAccData ACCESS ADR(bUIMagAccData);
	pa_tyProdRcpList ACCESS ADR(a_tyProdRcpList);
	p_tyCurrProdRcp ACCESS ADR(tyCurrProdRcp);
	p_tyDispProdRcp ACCESS ADR(tyDispProdRcp);
	p_sCurrMagRcpNm ACCESS ADR(sCurrMagRcpNm);
	p_eTimeStat ACCESS ADR(eTimeStat);
	p_eTimeStatus ACCESS ADR(eTimeStatus);
	p_bAccNewRcpCond ACCESS ADR(bAccNewRcpCond);
	p_bUpdtNewRcpCond ACCESS ADR(bUpdtNewRcpCond);
	p_bAutoUpdtData ACCESS ADR(bAutoUpdtData);
	p_sInfoMsg ACCESS ADR(sInfoMsg);
	p_bInternalUse ACCESS ADR(bInternalUse);
	p_tyInternalReqProdRcp ACCESS ADR(tyInternalReqProdRcp);
	p_bNewBrdEnteredCond ACCESS ADR(bNewBrdEnteredCond);
	p_bOldBrdExitedCond ACCESS ADR(bOldBrdExitedCond);
	p_bRlsBrd ACCESS ADR(bRlsBrd);
	p_tyToLeaderProdRcp ACCESS ADR(tyToLeaderProdRcp);
	p_bInternalReqProdRcpDiff ACCESS ADR(bInternalReqProdRcpDiff);
	p_bUpdtProdRcpDiff ACCESS ADR(bUpdtProdRcpDiff);
	p_bRlsBrdProdRcpDiff ACCESS ADR(bRlsBrdProdRcpDiff);
	p_sProgNm ACCESS ADR(sProgNm);
	p_bNtSettingsLoadDone ACCESS ADR(bNtSettingsLoadDone);
	p_tOnlineChkDlyTm ACCESS ADR(tOnlineChkDlyTm);
	p_bManual ACCESS ADR(bManual);
	p_bErr ACCESS ADR(bErr);
	p_bWarning ACCESS ADR(bWarning);
	p_bOps ACCESS ADR(bOps);
	p_bStandby ACCESS ADR(bStandby);
	p_eAWStat ACCESS ADR(eAWStat);
	p_bWidth2Prep ACCESS ADR(bWidth2Prep);
	p_bDBAOnWOAlign ACCESS ADR(bDBAOnWOAlign);

END_ACTION
```
